Universal Robots PolyScope program: Presentacion.urp

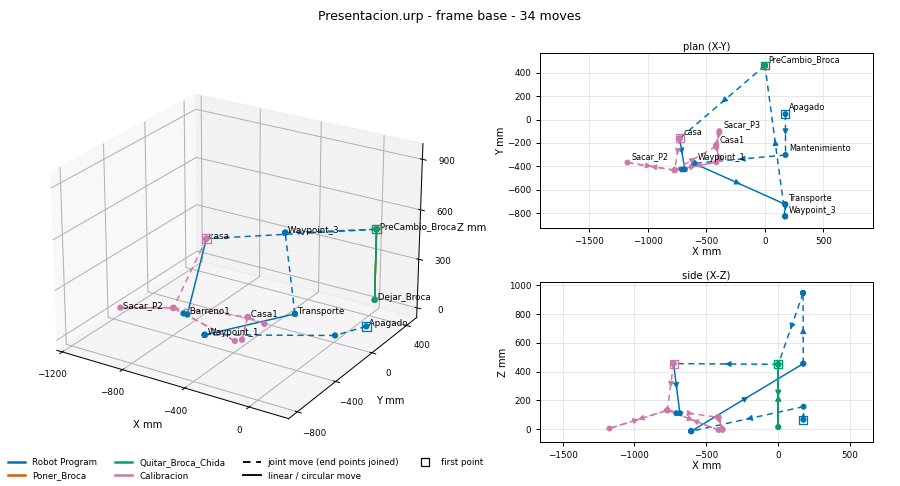
[picture p0: tool path of Presentacion.urp in frame base, 34 of 69 moves have a stored position in this frame; points joined in program order, loops and branches not executed]
Program Presentacion (installation=instalacion_derecha_10_MAR_21 directory=/programs/Presentacion createdIn=5.6.0.90886 lastSavedIn=5.6.0.90886 robotSerialNumber=20195001785)
Calibrated DH parameters: a=[0.000107, -0.568984, -0.552934, -0.00001, -0.000063, 0]; d=[0.180718, -257.998067, 200.685024, 57.48776, 0.119923, 0.115353]; alpha=[1.571119, 0.000876, -0.002498, 1.571178, -1.570523, 0]; deltaTheta=[0, -0.378191, 0.631587, -0.253396, 0, 0]
Robot Program (runOnlyOnce=false)
  MoveJ speed 60 deg/s, acceleration 80 deg/s^2 (useActiveTCP=true) feature=Base
    Waypoint Apagado: TCP in base x=175.753 y=46.675 z=64.304 mm, rx=-1.7747 ry=0.1396 rz=0.1139 rad; joints [90.002, -90.002, 153.585, 15, 89.999, 0.002] deg; TCP offset x=0.411 y=-218.298 z=37.994 mm, rx=1.558 ry=-0.1255 rz=0.1212 rad
    Waypoint Mantenimiento: TCP in base x=176.923 y=-302.82 z=155.559 mm, rx=0.3579 ry=-0.0299 rz=0.1455 rad; joints [90.14, -9.678, 128.928, 81.812, 89.499, -0.139] deg; TCP offset x=0.411 y=-218.298 z=37.994 mm, rx=1.558 ry=-0.1255 rz=0.1212 rad
  Folder Variables
    muestras := 3
    muestrasTomadas := 0
    alpha := 0
    P1 := p[0,0,0,0,0,0]
    P2 := p[0,0,0,0,0,0]
    P3 := p[0,0,0,0,0,0]
    P4 := p[0,0,0,0,0,0]
    Coordenada := p[0,0,0,0,0,0]
    MoveJ speed 60 deg/s, acceleration 80 deg/s^2 (useActiveTCP=true) feature=Base
      Loop Forever
        Waypoint Waypoint_1: TCP in base x=-604.792 y=-374.483 z=-15.265 mm, rx=2.0075 ry=-2.3999 rz=-0.0198 rad; joints [22.691, -71.513, 121.887, -50.957, 113.675, -0.127] deg; TCP offset x=0.411 y=-218.298 z=37.994 mm, rx=1.558 ry=-0.1255 rz=0.1212 rad
        Waypoint Waypoint_2: TCP in base x=-604.92 y=-374.48 z=-15.28 mm, rx=2.0074 ry=-2.4 rz=-0.0198 rad; joints [22.686, -71.504, 121.876, -50.954, 113.672, -0.127] deg
        var_7 := pose_dist(Waypoint_1, Waypoint_2)
      Waypoint Waypoint_1 referenceName=Waypoint_1: TCP in base x=-604.792 y=-374.483 z=-15.265 mm, rx=2.0075 ry=-2.3999 rz=-0.0198 rad; joints [22.691, -71.513, 121.887, -50.957, 113.675, -0.127] deg
      Waypoint Waypoint_2 referenceName=Waypoint_2: TCP in base x=-604.92 y=-374.48 z=-15.28 mm, rx=2.0074 ry=-2.4 rz=-0.0198 rad; joints [22.686, -71.504, 121.876, -50.954, 113.672, -0.127] deg
    pch_atual := get_actual_tcp_pose()
    Popup Message (haltProgram=false message=hi inputType=Variable) variable=pch_atual
  Folder Movimiento eje 7
    MoveL speed 250 mm/s, acceleration 1200 mm/s^2 (useActiveTCP=true) feature=Base
      Waypoint Transporte: TCP in base x=174.984 y=-724.59 z=455.169 mm, rx=3.1229 ry=-0.2484 rz=-0.0011 rad; joints [90, -90.004, 90.001, 0, 90, 0] deg; TCP offset x=0.411 y=-218.298 z=37.994 mm, rx=1.558 ry=-0.1255 rz=0.1212 rad
      Set DigitalOutput pin=postrnas_m187; digitalValue=1
      SuppressedNode
        Set ExpressionOutput pin=pos_2_mw3; expression=2
      num_barreno := str_cat("Barreno: ",1)
      var_6 := get_actual_tcp_pose()
      X_actual := str_cat("     X: ",var_6[0])
      Y_actual := str_cat("     Y: ",var_6[1])
      pos_barreno := str_cat(X_actual,Y_actual)
      Script: textmsg("------------------DAS LOG------------------")
      Script: textmsg(num_barreno,pos_barreno)
      Popup Warning (haltProgram=false message=hsjd inputType=Text)
  Folder Saludos
    MoveL speed 250 mm/s, acceleration 1200 mm/s^2 (useActiveTCP=true) feature=Base
      Waypoint Transporte: TCP in base x=174.984 y=-724.59 z=455.169 mm, rx=3.1229 ry=-0.2484 rz=-0.0011 rad; joints [90, -90.004, 90.001, 0, 90, 0] deg
      Set DigitalOutput pin=postrnas_m187; digitalValue=1
      SuppressedNode
        MoveJ speed 60 deg/s, acceleration 80 deg/s^2 (useActiveTCP=true) feature=Base
          Waypoint Casa: TCP in base x=728.924 y=-154.439 z=454.335 mm, rx=2.3654 ry=2.0675 rz=0 rad; joints [1.567, -90.267, -89.594, -180.639, -89.764, 0.039] deg
      MoveJ speed 60 deg/s, acceleration 80 deg/s^2 (useActiveTCP=true) feature=Base
        SuppressedNode
          Waypoint Waypoint_1: TCP in base x=65.093 y=-826.886 z=901.889 mm, rx=1.4338 ry=-0.7424 rz=0.7302 rad; joints [89.992, -97.74, 97.176, -89.444, 134.994, 0.001] deg
        Set DigitalOutput pin=postrnas_m187; digitalValue=0
        Waypoint Waypoint_3: TCP in base x=173.453 y=-827.062 z=946.896 mm, rx=1.4805 ry=-0.6168 rz=0.6108 rad; joints [98.118, -94.832, 92.691, -93.201, 125.502, -9.597] deg
        SuppressedNode
          Waypoint Waypoint_5: TCP in base x=173.423 y=-741.68 z=946.84 mm, rx=1.2989 ry=-0.7251 rz=0.6034 rad; joints [102.47, -97.376, 99.801, -114.266, 126.347, -24.689] deg
      Loop Counting (count=15) loopVariable(name=Loop_1)
        MoveL speed 1500 mm/s, acceleration 2200 mm/s^2 (useActiveTCP=true) feature=Base
          SuppressedNode
            Waypoint Waypoint_1: motionParameters(blendRadius=0.05); TCP in base x=65.093 y=-826.886 z=901.889 mm, rx=1.4338 ry=-0.7424 rz=0.7302 rad; joints [89.992, -97.74, 97.176, -89.444, 134.994, 0.001] deg
          SuppressedNode
            Waypoint Waypoint_2: motionParameters(blendRadius=0.05); TCP in base x=281.914 y=-909.743 z=901.9 mm, rx=1.5058 ry=0.4887 rz=-0.49 rad; joints [89.998, -90.003, 89.996, -90, 45, 0.004] deg
          Waypoint Waypoint_3: TCP in base x=173.453 y=-827.062 z=946.896 mm, rx=1.4805 ry=-0.6168 rz=0.6108 rad; joints [98.118, -94.832, 92.691, -93.201, 125.502, -9.597] deg
          Waypoint Waypoint_4: TCP in base x=173.444 y=-827.101 z=946.817 mm, rx=1.4837 ry=0.6112 rz=-0.6169 rad; joints [78.227, -99.572, 95.233, -100.465, 37.264, 18.965] deg
          SuppressedNode
            Waypoint Waypoint_5: motionParameters(jointSpeed=1.047198 jointAcceleration=1.396263 cartesianSpeed=0.25 cartesianAcceleration=1.2); TCP in base x=173.423 y=-741.68 z=946.84 mm, rx=1.2989 ry=-0.7251 rz=0.6034 rad; joints [102.47, -97.376, 99.801, -114.266, 126.347, -24.689] deg
          SuppressedNode
            Waypoint Waypoint_6: motionParameters(jointSpeed=1.047198 jointAcceleration=1.396263 cartesianSpeed=0.25 cartesianAcceleration=1.2); TCP in base x=173.459 y=-827.104 z=946.825 mm, rx=1.6228 ry=0.6313 rz=-0.7589 rad; joints [80.134, -100.807, 88.516, -73.712, 30.209, 3.288] deg
        SuppressedNode
          Waypoint Waypoint_1: TCP in base x=-291.405 y=-499.146 z=911.663 mm, rx=1.27 ry=-0.6711 rz=0.7685 rad; joints [-90.912, -52.098, -119.496, -88.535, -44.817, 0.182] deg
        SuppressedNode
          Waypoint Waypoint_2: TCP in base x=-77.693 y=-536.254 z=818.128 mm, rx=1.4537 ry=0.4411 rz=-0.4893 rad; joints [-90.912, -53.514, -125.158, -87.62, -133.489, 0.185] deg
      Popup Message (haltProgram=false message=arranquesito inputType=Text)
  SuppressedNode
    Popup Message (haltProgram=false message=opsjd inputType=Text)
  SuppressedNode
    Folder Paro_Emergencia
      MoveJ speed 60 deg/s, acceleration 80 deg/s^2 (useActiveTCP=true) feature=Base
        Waypoint Waypoint_3: TCP in base x=-687.031 y=180.786 z=3.5 mm, rx=1.8753 ry=-2.5169 rz=0.0061 rad; joints [-178.733, -104.887, -123.784, -131.854, -81.244, 0.422] deg
      MoveL speed 250 mm/s, acceleration 1200 mm/s^2 (useActiveTCP=true) feature=Base
        Loop Forever
          Waypoint Waypoint_3: TCP in base x=-687.031 y=180.786 z=3.5 mm, rx=1.8753 ry=-2.5169 rz=0.0061 rad; joints [-178.733, -104.887, -123.784, -131.854, -81.244, 0.422] deg
          Waypoint Waypoint_4: TCP in base x=-687.031 y=-113.957 z=3.5 mm, rx=1.8753 ry=-2.5169 rz=0.0061 rad; joints [-147.777, -104.253, -124.677, -131.662, -50.29, 0.749] deg
  Folder Cambio_Brocas
    Loop Counting (count=1) loopVariable=Loop_1
      MoveJ speed 60 deg/s, acceleration 80 deg/s^2 (useActiveTCP=true) feature=Base
        SuppressedNode
          Waypoint Transporte: TCP in base x=174.984 y=-724.59 z=455.169 mm, rx=3.1229 ry=-0.2484 rz=-0.0011 rad; joints [90, -90.004, 90.001, 0, 90, 0] deg
        SuppressedNode
          Waypoint Casa: TCP in base x=728.924 y=-154.439 z=454.335 mm, rx=2.3654 ry=2.0675 rz=0 rad; joints [1.567, -90.267, -89.594, -180.639, -89.764, 0.039] deg
        SuppressedNode
          Waypoint Pre_Casa: TCP in base x=724.591 y=175.02 z=455.143 mm, rx=2.3854 ry=2.034 rz=0.009 rad; joints [180.002, -90.001, 89.999, 0.004, 90, 0.002] deg; TCP offset x=0.411 y=-218.298 z=37.994 mm, rx=1.558 ry=-0.1255 rz=0.1212 rad
        SuppressedNode
          Waypoint Waypoint_7: TCP in base x=327.444 y=571.558 z=453.852 mm, rx=2.3843 ry=2.0357 rz=0.0036 rad; joints [90, -90, -90, -180, 0, 0] deg; TCP offset x=0.411 y=-218.298 z=37.994 mm, rx=1.558 ry=-0.1255 rz=0.1212 rad
        Waypoint PreCambio_Broca: TCP in base x=0.946 y=461.694 z=450 mm, rx=-0.2787 ry=-3.1292 rz=0 rad; joints [124.465, -59.781, -112.137, -188.57, -54.361, 0.335] deg
        SuppressedNode
          Loop Counting (count=50) loopVariable(name=Loop_1)
            Call Poner_Broca
            Call Quitar_Broca_Chida
        Call Poner_Broca
  Folder Barrenado
    alpha := 0
    Loop Forever
      MoveJ speed 60 deg/s, acceleration 80 deg/s^2 (useActiveTCP=true) feature=Base
        Waypoint casa: TCP in base x=-727.761 y=-161.288 z=455.169 mm, rx=2.012 ry=-2.4053 rz=-0.0107 rad; joints [-1.081, -90.004, 90.001, 0, 90, 0] deg; TCP offset x=0.411 y=-218.298 z=37.994 mm, rx=1.558 ry=-0.1255 rz=0.1212 rad
        Call Calibracion
        Call GoNoGo
        MoveL speed 250 mm/s, acceleration 1200 mm/s^2 (useActiveTCP=true) feature=Base
          Waypoint Barreno1: TCP in base x=-683.897 y=-425.831 z=110.04 mm, rx=3.0978 ry=-0.4471 rz=-0.0122 rad; joints [216.485, -110.43, -101.989, -147.498, -136.182, -0.299] deg
          Waypoint Barreno2: TCP in base x=-709.31 y=-425.852 z=110.052 mm, rx=3.0978 ry=-0.4471 rz=-0.0123 rad; joints [215.28, -112.388, -99.127, -148.4, -137.383, -0.296] deg
          Loop Counting (count=2) loopVariable(name=Loop_9)
            If alpha≤16
              internos := interpolate_pose(Barreno1, Barreno2, alpha)
              bajada := p[0,0,-0.024,0,0,0]
              subida := p[0,0,0.024,0,0,0]
              Waypoint Waypoint (Variable): variable=internos
              MoveDirectionNode (selectedDirection=ZMinus)
                Until DISTANCE (allowActions=false deceleration=3 distanceNodeType=STOP) Distance=0.067; motionParameters(blendRadius=0)
              MoveDirectionNode (selectedDirection=ZMinus toolParams=0.0013, 2.0E-4)
                Until TOOL_CONTACT_DETECTION (allowActions=false retraction=0 decelerationAcceleration=9 decelerationAngularAcceleration=34.906585)
              Wait Sleep waitTime=0.3
              Set DigitalOutput pin=config_out[1]; digitalValue=1
              Wait Sleep waitTime=0.5
              Set DigitalOutput pin=config_out[1]; digitalValue=0
              MoveDirectionNode (selectedDirection=ZPlus)
                Until DISTANCE (allowActions=false deceleration=3 distanceNodeType=STOP) Distance=0.002; motionParameters(blendRadius=0)
              Wait Sleep waitTime=0.5
              Set DigitalOutput pin=config_out[1]; digitalValue=1
              Wait Sleep waitTime=0.3
              Loop Counting (count=1) loopVariable(name=Loop_6)
                bajar := pose_add(get_actual_tcp_pose(), bajada)
                Waypoint Waypoint (Variable): motionParameters(jointSpeed=1.047198 jointAcceleration=1.396263 cartesianSpeed=0.005 cartesianAcceleration=0.01); variable=bajar
                subir := pose_add(get_actual_tcp_pose(), subida)
                Waypoint Waypoint (Variable): motionParameters(jointSpeed=1.047198 jointAcceleration=1.396263 cartesianSpeed=0.02 cartesianAcceleration=0.02); variable=subir
                bajada := pose_add(bajada, p[0,0,-0.008,0,0,0])
                subida := pose_add(subida, p[0,0,0.008,0,0,0])
              Set DigitalOutput pin=config_out[1]; digitalValue=0
              MoveDirectionNode (selectedDirection=ZPlus)
                Until DISTANCE (allowActions=false deceleration=3 distanceNodeType=STOP) Distance=0.1; motionParameters(blendRadius=0)
              alpha := alpha+1
            Else 
              Popup Message (haltProgram=false message=linea barrenada inputType=Text)
              Call Quitar_Broca_Chida
              Popup Message (haltProgram=false message=fin inputType=Text)
        Call Quitar_Broca_Chida
        Call Poner_Broca
SubProgram -> Poner_Broca
SubProgram -> Quitar_Broca_Chida
SubProgram -> Calibracion
SubProgram -> GoNoGo
SubProgram Poner_Broca (keepSynchronizedWithDisk=false)
  Folder Poner_Broca
    Set DigitalOutput pin=ini_cambro_m289; digitalValue=0
    MoveL speed 250 mm/s, acceleration 1200 mm/s^2 (useActiveTCP=true) feature=Base
      Waypoint PreCambio_Broca: TCP in base x=0.946 y=461.694 z=450 mm, rx=-0.2787 ry=-3.1292 rz=0 rad; joints [124.465, -59.781, -112.137, -188.57, -54.361, 0.335] deg; TCP offset x=0.411 y=-218.298 z=37.994 mm, rx=1.558 ry=-0.1255 rz=0.1212 rad
      Waypoint Dejar_Broca: TCP in base x=0.946 y=461.694 z=13.784 mm, rx=-0.2787 ry=-3.1292 rz=0 rad; joints [124.423, -78.567, -149.823, -132.118, -54.538, 0.369] deg; TCP offset x=0.411 y=-218.298 z=37.994 mm, rx=1.558 ry=-0.1255 rz=0.1212 rad
    Set DigitalOutput pin=ini_cambro_m289; digitalValue=1
    Wait Sleep waitTime=3.8
    Set DigitalOutput pin=ini_cambro_m289; digitalValue=0
    Wait Sleep waitTime=0.5
    Wait DigitalInput pin=fciclocarr_m292; digitalValue=0
    Wait Sleep waitTime=0.5
    MoveL speed 250 mm/s, acceleration 1200 mm/s^2 (useActiveTCP=true) feature=Base
      Waypoint PreCambio_Broca: TCP in base x=0.946 y=461.694 z=450 mm, rx=-0.2787 ry=-3.1292 rz=0 rad; joints [124.465, -59.781, -112.137, -188.57, -54.361, 0.335] deg; TCP offset x=0.411 y=-218.298 z=37.994 mm, rx=1.558 ry=-0.1255 rz=0.1212 rad
      SuppressedNode
        MoveJ speed 60 deg/s, acceleration 80 deg/s^2 (useActiveTCP=true) feature=Base
          Waypoint casa: TCP in base x=-327.476 y=-571.536 z=453.871 mm, rx=2.0383 ry=-2.3875 rz=-0.0101 rad; joints [269.996, -89.998, -90, -179.999, 0, 0] deg; TCP offset x=0.411 y=-218.298 z=37.994 mm, rx=1.558 ry=-0.1255 rz=0.1212 rad
    SuppressedNode
      Popup Message (haltProgram=false message=kon inputType=Text)
SubProgram Quitar_Broca_Chida (keepSynchronizedWithDisk=false)
  Folder Quitar_Broca
    MoveJ speed 60 deg/s, acceleration 80 deg/s^2 (useActiveTCP=true) feature=Base
      SuppressedNode
        Waypoint casa: TCP in base x=-734.526 y=-232.925 z=166.215 mm, rx=3.0978 ry=-0.4471 rz=-0.0122 rad; joints [200.498, -107.87, -99.095, -152.973, -152.157, -0.273] deg
      Loop Counting (count=1) loopVariable(name=Loop_3)
        MoveL speed 250 mm/s, acceleration 1200 mm/s^2 (useActiveTCP=true) feature=Base
          SuppressedNode
            MoveJ speed 60 deg/s, acceleration 80 deg/s^2 (useActiveTCP=true) feature=Base
              Waypoint casa: TCP in base x=-327.476 y=-571.536 z=453.871 mm, rx=2.0383 ry=-2.3875 rz=-0.0101 rad; joints [269.996, -89.998, -90, -179.999, 0, 0] deg
          MoveDirectionNode (selectedDirection=ZPlus)
            Until DISTANCE (allowActions=false deceleration=3 distanceNodeType=STOP) Distance=0.1; motionParameters(blendRadius=0)
          MoveJ speed 60 deg/s, acceleration 80 deg/s^2 (useActiveTCP=true) feature=Base
            Waypoint PreCambio_Broca: TCP in base x=0.946 y=461.694 z=450 mm, rx=-0.2787 ry=-3.1292 rz=0 rad; joints [124.465, -59.781, -112.137, -188.57, -54.361, 0.335] deg; TCP offset x=0.411 y=-218.298 z=37.994 mm, rx=1.558 ry=-0.1255 rz=0.1212 rad
          Waypoint Dejar_Broca: motionParameters(jointSpeed=1.047198 jointAcceleration=1.396263 cartesianSpeed=0.15 cartesianAcceleration=0.2); TCP in base x=0.946 y=461.694 z=13.784 mm, rx=-0.2787 ry=-3.1292 rz=0 rad; joints [124.423, -78.567, -149.823, -132.118, -54.538, 0.369] deg; TCP offset x=0.411 y=-218.298 z=37.994 mm, rx=1.558 ry=-0.1255 rz=0.1212 rad
          Set DigitalOutput pin=outputbroc_m291; digitalValue=1
          Wait Sleep waitTime=0.5
          Set DigitalOutput pin=outputbroc_m291; digitalValue=0
          Wait Sleep waitTime=0.5
          Wait DigitalInput pin=fciclocarr_m292; digitalValue=0
          Wait Sleep waitTime=0.5
          SuppressedNode
            MoveDirectionNode (selectedDirection=ZPlus)
              Until DISTANCE (allowActions=false deceleration=3 distanceNodeType=STOP) Distance=0.5; motionParameters(blendRadius=0)
          Waypoint PreCambio_Broca: TCP in base x=0.946 y=461.694 z=450 mm, rx=-0.2787 ry=-3.1292 rz=0 rad; joints [124.465, -59.781, -112.137, -188.57, -54.361, 0.335] deg; TCP offset x=0.411 y=-218.298 z=37.994 mm, rx=1.558 ry=-0.1255 rz=0.1212 rad
          Set DigitalOutput pin=avancarrusel_m7; digitalValue=1
          Wait Sleep waitTime=1.1
          Set DigitalOutput pin=avancarrusel_m7; digitalValue=0
          SuppressedNode
            Popup Message (haltProgram=false message=kon inputType=Text)
SubProgram Calibracion (keepSynchronizedWithDisk=false)
  Folder Calibracion
    Folder Subvariables
      muestras := 1
      muestrasTomadas := 0
      P1 := p[0,0,0,0,0,0]
      P2 := p[0,0,0,0,0,0]
      P3 := p[0,0,0,0,0,0]
      P4 := p[0,0,0,0,0,0]
      rotaciones := p[0,0,0,0,0,0]
      PosFinal := p[0,0,0,0,0,0]
      m1 := 0
      m2 := 0
      b1 := 0
      b2 := 0
      Xd := 0
      Yd := 0
      Xp := 0
      Yp := 0
      Xfin := 0
      Yfin := 0
    SuppressedNode
      Folder plano mod
        Loop Forever
          MoveL speed 250 mm/s, acceleration 1200 mm/s^2 (useActiveTCP=true) feature=Plane_5
            Popup Message (haltProgram=false inputType=Variable) variable(featureName=Plane_5)
            Waypoint Waypoint_5: TCP in base x=-413.934 y=-364.729 z=55.217 mm, rx=2.0101 ry=-2.4031 rz=-0.0102 rad; joints [31.806, -89.454, 133.906, -44.626, 122.803, 0.104] deg; TCP offset x=0.411 y=-218.298 z=37.994 mm, rx=1.558 ry=-0.1255 rz=0.1212 rad; feature pose in base x=-414.632 y=-364.771 z=-8.601 mm, rx=0.0051 ry=-3.1307 rz=0.001 rad
            Waypoint Waypoint_6: TCP in base x=-770.877 y=-364.729 z=55.217 mm, rx=2.0101 ry=-2.4031 rz=-0.0102 rad; joints [16.666, -66.533, 104.244, -37.849, 107.67, 0.156] deg
            SuppressedNode
              Script: 
            Script file /programs/Presentacion/nivelacion.script
              | MoveJ
              |       Waypoint_5
              | 
              | Plane5_const = pose_trans(Plane5_const, p[-0.5,-0.25,0.1,2.010,-2.403,-0.010])
            Popup Message (haltProgram=false inputType=Variable) variable(featureName=Plane_5)
            Waypoint Waypoint_5: TCP in base x=-413.934 y=-364.729 z=55.217 mm, rx=2.0101 ry=-2.4031 rz=-0.0102 rad; joints [31.806, -89.454, 133.906, -44.626, 122.803, 0.104] deg
            Waypoint Waypoint_6: TCP in base x=-770.877 y=-364.729 z=55.217 mm, rx=2.0101 ry=-2.4031 rz=-0.0102 rad; joints [16.666, -66.533, 104.244, -37.849, 107.67, 0.156] deg
    Folder Nivelacion
      SuppressedNode
        MoveL speed 250 mm/s, acceleration 1200 mm/s^2 (useActiveTCP=true) feature=Base
          MoveDirectionNode (selectedDirection=ZPlus)
            Until DISTANCE (allowActions=false deceleration=3 distanceNodeType=STOP) Distance=0.1; motionParameters(blendRadius=0)
          MoveJ speed 60 deg/s, acceleration 80 deg/s^2 (useActiveTCP=true) feature=Base
            Waypoint casa: TCP in base x=-727.761 y=-161.288 z=455.169 mm, rx=2.012 ry=-2.4053 rz=-0.0107 rad; joints [-1.081, -90.004, 90.001, 0, 90, 0] deg; TCP offset x=0.411 y=-218.298 z=37.994 mm, rx=1.558 ry=-0.1255 rz=0.1212 rad
          MoveL speed 250 mm/s, acceleration 1200 mm/s^2 (useActiveTCP=true) feature=Base
            MoveJ speed 60 deg/s, acceleration 80 deg/s^2 (useActiveTCP=true) feature=Base
              Waypoint Casa2: TCP in base x=-771.172 y=-432.935 z=130.553 mm, rx=2.0075 ry=-2.3998 rz=-0.0199 rad; joints [21.893, -67.533, 96.816, -29.884, 112.905, -0.164] deg
            Folder P1
              Loop While (checkContinuously=false) expression=muestrasTomadas<muestras
                MoveJ speed 60 deg/s, acceleration 80 deg/s^2 (useActiveTCP=true) feature=Base
                  Waypoint Sacar_P1: motionParameters(jointSpeed=1.047198 jointAcceleration=1.396263 cartesianSpeed=0.1 cartesianAcceleration=0.15); TCP in base x=-414.596 y=-364.737 z=-6.973 mm, rx=2.0075 ry=-2.3998 rz=-0.0199 rad; joints [31.933, -83.207, 136.677, -54.117, 122.913, -0.246] deg; TCP offset x=0.411 y=-218.298 z=37.994 mm, rx=1.558 ry=-0.1255 rz=0.1212 rad
                  SuppressedNode
                    Waypoint Sacar_P5: TCP in base x=-414.62 y=-364.74 z=-8.63 mm, rx=2.0074 ry=-2.3998 rz=-0.0199 rad; joints [31.932, -83.024, 136.735, -54.36, 122.914, -0.245] deg
                Wait Sleep waitTime=0.5
                MoveDirectionNode (selectedDirection=ZMinus toolParams=0.0013, 2.0E-4)
                  Until TOOL_CONTACT_DETECTION (allowActions=false retraction=0 decelerationAcceleration=9 decelerationAngularAcceleration=34.906585)
                Wait Sleep waitTime=2
                P5 := pose_add(get_actual_tcp_pose(), P5)
                muestrasTomadas := muestrasTomadas+1
              muestrasTomadas := 0
              var_1 := (P5[0])/muestras
              var_2 := (P5[1])/muestras
              var_8 := (P5[2])/muestras
              rotaciones := get_actual_tcp_pose()
              var_3 := rotaciones[3]
              var_4 := rotaciones[4]
              var_5 := rotaciones[5]
              P5 := p[var_1,var_2,var_8,var_3,var_4,var_5]
            MoveJ speed 60 deg/s, acceleration 80 deg/s^2 (useActiveTCP=true) feature=Base
              Waypoint Casa2: TCP in base x=-771.172 y=-432.935 z=130.553 mm, rx=2.0075 ry=-2.3998 rz=-0.0199 rad; joints [21.893, -67.533, 96.816, -29.884, 112.905, -0.164] deg; TCP offset x=0.411 y=-218.298 z=37.994 mm, rx=1.558 ry=-0.1255 rz=0.1212 rad
            Folder P2
              Loop While (checkContinuously=false) expression=muestrasTomadas<muestras
                MoveJ speed 60 deg/s, acceleration 80 deg/s^2 (useActiveTCP=true) feature=Base
                  Waypoint Sacar_P2: TCP in base x=-1173.98 y=-367.222 z=3.642 mm, rx=2.0075 ry=-2.3998 rz=-0.0199 rad; joints [10.692, -31.748, 48.291, -17.094, 101.74, -0.036] deg; TCP offset x=0.411 y=-218.298 z=37.994 mm, rx=1.558 ry=-0.1255 rz=0.1212 rad
                  SuppressedNode
                    Waypoint Sacar_P6: TCP in base x=-1173.985 y=-367.26 z=-0.32 mm, rx=2.0075 ry=-2.3998 rz=-0.0199 rad; joints [10.694, -31.605, 48.427, -17.374, 101.738, -0.036] deg
                Wait Sleep waitTime=0.5
                MoveDirectionNode (selectedDirection=YPlus toolParams=0.0013, 2.0E-4)
                  Until TOOL_CONTACT_DETECTION (allowActions=false retraction=0 decelerationAcceleration=9 decelerationAngularAcceleration=34.906585)
                Wait Sleep waitTime=2
                P2 := pose_add(get_actual_tcp_pose(), P2)
                muestrasTomadas := muestrasTomadas+1
              muestrasTomadas := 0
              var_1 := (P2[0])/muestras
              var_2 := (P2[1])/muestras
              rotaciones := get_actual_tcp_pose()
              var_3 := rotaciones[3]
              var_4 := rotaciones[4]
              var_5 := rotaciones[5]
              P2 := p[var_1,var_2,-0.37,var_3,var_4,var_5]
            MoveJ speed 60 deg/s, acceleration 80 deg/s^2 (useActiveTCP=true) feature=Base
              Waypoint Casa2: TCP in base x=-771.172 y=-432.935 z=130.553 mm, rx=2.0075 ry=-2.3998 rz=-0.0199 rad; joints [21.893, -67.533, 96.816, -29.884, 112.905, -0.164] deg; TCP offset x=0.411 y=-218.298 z=37.994 mm, rx=1.558 ry=-0.1255 rz=0.1212 rad
            Folder m1
              var_1 := (P1[0])
              var_2 := (P1[1])
              var_3 := (P2[0])
              var_4 := (P2[1])
              m1 := (var_4-var_2)/(var_3-var_1)
            Folder b1
              b1 := ((m1*var_1)-var_2)*(-1)
            MoveJ speed 60 deg/s, acceleration 80 deg/s^2 (useActiveTCP=true) feature=Base
              Waypoint Casa1: TCP in base x=-397.714 y=-209.387 z=130.553 mm, rx=2.0075 ry=-2.3998 rz=-0.0199 rad; joints [8.28, -111.842, 141.427, -30.137, 99.306, -0.058] deg; TCP offset x=0.411 y=-218.298 z=37.994 mm, rx=1.558 ry=-0.1255 rz=0.1212 rad
            Folder P3
              Loop While (checkContinuously=false) expression=muestrasTomadas<muestras
                MoveJ speed 60 deg/s, acceleration 80 deg/s^2 (useActiveTCP=true) feature=Base
                  Waypoint Sacar_P3: motionParameters(jointSpeed=1.047198 jointAcceleration=1.396263 cartesianSpeed=0.1 cartesianAcceleration=0.15); TCP in base x=-389.257 y=-99.052 z=-5.952 mm, rx=2.0075 ry=-2.3998 rz=-0.0199 rad; joints [-19.785, -107.959, 157.177, -49.758, 71.211, 0.249] deg
                  SuppressedNode
                    Waypoint Sacar_P7: TCP in base x=-389.26 y=-99.06 z=-9.06 mm, rx=2.0075 ry=-2.3998 rz=-0.02 rad; joints [-19.783, -107.388, 157.374, -50.532, 71.212, 0.252] deg
                Wait Sleep waitTime=0.5
                MoveDirectionNode (selectedDirection=XPlus toolParams=0.0013, 2.0E-4)
                  Until TOOL_CONTACT_DETECTION (allowActions=false retraction=0 decelerationAcceleration=9 decelerationAngularAcceleration=34.906585)
                Wait Sleep waitTime=2
                P3 := pose_add(get_actual_tcp_pose(), P3)
                muestrasTomadas := muestrasTomadas+1
              muestrasTomadas := 0
              var_1 := (P3[0])/muestras
              var_2 := (P3[1])/muestras
              rotaciones := get_actual_tcp_pose()
              var_3 := rotaciones[3]
              var_4 := rotaciones[4]
              var_5 := rotaciones[5]
              P3 := p[var_1,var_2,-0.37,var_3,var_4,var_5]
            MoveJ speed 60 deg/s, acceleration 80 deg/s^2 (useActiveTCP=true) feature=Base
              Waypoint Casa1: TCP in base x=-397.714 y=-209.387 z=130.553 mm, rx=2.0075 ry=-2.3998 rz=-0.0199 rad; joints [8.28, -111.842, 141.427, -30.137, 99.306, -0.058] deg
            Folder P4
              Loop While (checkContinuously=false) expression=muestrasTomadas<muestras
                MoveJ speed 60 deg/s, acceleration 80 deg/s^2 (useActiveTCP=true) feature=Base
                  Waypoint Sacar_P4: motionParameters(jointSpeed=1.047198 jointAcceleration=1.396263 cartesianSpeed=0.1 cartesianAcceleration=0.15); TCP in base x=-387.922 y=-336.637 z=-4.002 mm, rx=2.0075 ry=-2.3998 rz=-0.0199 rad; joints [30.437, -87.075, 140.636, -54.198, 121.418, -0.23] deg
                Wait Sleep waitTime=0.5
                MoveDirectionNode (selectedDirection=XPlus toolParams=0.0013, 2.0E-4)
                  Until TOOL_CONTACT_DETECTION (allowActions=false retraction=0 decelerationAcceleration=9 decelerationAngularAcceleration=34.906585)
                Wait Sleep waitTime=2
                P4 := pose_add(get_actual_tcp_pose(), P4)
                muestrasTomadas := muestrasTomadas+1
              muestrasTomadas := 0
              var_1 := (P4[0])/muestras
              var_2 := (P4[1])/muestras
              rotaciones := get_actual_tcp_pose()
              var_3 := rotaciones[3]
              var_4 := rotaciones[4]
              var_5 := rotaciones[5]
              P4 := p[var_1,var_2,-0.37,var_3,var_4,var_5]
            MoveJ speed 60 deg/s, acceleration 80 deg/s^2 (useActiveTCP=true) feature=Base
              Waypoint Casa1: TCP in base x=-397.714 y=-209.387 z=130.553 mm, rx=2.0075 ry=-2.3998 rz=-0.0199 rad; joints [8.28, -111.842, 141.427, -30.137, 99.306, -0.058] deg
            Folder m2
              var_1 := (P3[0])
              var_2 := (P3[1])
              var_3 := (P4[0])
              var_4 := (P4[1])
              m2 := (var_4-var_2)/(var_3-var_1)
            Folder b2
              b2 := ((m2*var_1)-var_2)*(-1)
            Folder Xd y Yd
              Xd := (b2-b1)/(m1-m2)
              Yd := (m1*Xd)+b1
            Folder Xp y Yp
              Xp := (1)/(sqrt((m1*m1)+1))
              Yp := (m2)/(sqrt((m2*m2)+1))
            Folder Origen
              Xfin := ((0*Xp)-(Xd)-(0*(1/m2)))*(-1)
              Yfin := ((0*Yp)-(Yd)+(0*m1))*(-1)
              rotaciones := get_actual_tcp_pose()
              var_3 := rotaciones[3]
              var_4 := rotaciones[4]
              var_5 := rotaciones[5]
              PosFinal := p[Xfin+0.00208915,Yfin+0.00208915,0.11,var_3,var_4,var_5]
            MoveJ speed 60 deg/s, acceleration 80 deg/s^2 (useActiveTCP=true) feature=Base
              Waypoint Waypoint (Variable): motionParameters(jointSpeed=1.047198 jointAcceleration=1.396263 cartesianSpeed=0.15 cartesianAcceleration=0.2); variable=PosFinal
            MoveDirectionNode (selectedDirection=ZPlus)
              Until DISTANCE (allowActions=false deceleration=3 distanceNodeType=STOP) Distance=0.1; motionParameters(blendRadius=0)
            MoveJ speed 60 deg/s, acceleration 80 deg/s^2 (useActiveTCP=true) feature=Base
              Waypoint Casa2: TCP in base x=-771.172 y=-432.935 z=130.553 mm, rx=2.0075 ry=-2.3998 rz=-0.0199 rad; joints [21.893, -67.533, 96.816, -29.884, 112.905, -0.164] deg; TCP offset x=0.411 y=-218.298 z=37.994 mm, rx=1.558 ry=-0.1255 rz=0.1212 rad
            Folder Linea1
              Folder Buje1
                Xfin := ((0.09525*Xp)-(Xd)-(-0.0127*(1/m2)))*(-1)
                Yfin := ((-0.0127*Yp)-(Yd)+(0.09525*m1))*(-1)
                rotaciones := get_actual_tcp_pose()
                var_3 := rotaciones[3]
                var_4 := rotaciones[4]
                var_5 := rotaciones[5]
                PosFinal := p[Xfin+0.00208915,Yfin+0.00208915,0.03,var_3,var_4,var_5]
                MoveL speed 250 mm/s, acceleration 1200 mm/s^2 (useActiveTCP=true) feature=Base
                  MoveJ speed 60 deg/s, acceleration 80 deg/s^2 (useActiveTCP=true) feature=Base
                    Waypoint Waypoint (Variable): motionParameters(jointSpeed=1.047198 jointAcceleration=1.396263 cartesianSpeed=0.15 cartesianAcceleration=0.2); variable=PosFinal
                  MoveDirectionNode (selectedDirection=ZMinus toolParams=0.02, 0.02)
                    Until DISTANCE (allowActions=false deceleration=3 distanceNodeType=STOP) Distance=0.035; motionParameters(blendRadius=0)
                  MoveDirectionNode (selectedDirection=ZPlus toolParams=0.02, 0.02)
                    Until DISTANCE (allowActions=false deceleration=3 distanceNodeType=STOP) Distance=0.035; motionParameters(blendRadius=0)
              Folder Buje2
                Xfin := ((0.12065*Xp)-(Xd)-(-0.0127*(1/m2)))*(-1)
                Yfin := ((-0.0127*Yp)-(Yd)+(0.12065*m1))*(-1)
                rotaciones := get_actual_tcp_pose()
                var_3 := rotaciones[3]
                var_4 := rotaciones[4]
                var_5 := rotaciones[5]
                PosFinal := p[Xfin+0.00208915,Yfin+0.00208915,0.03,var_3,var_4,var_5]
                MoveL speed 250 mm/s, acceleration 1200 mm/s^2 (useActiveTCP=true) feature=Base
                  MoveJ speed 60 deg/s, acceleration 80 deg/s^2 (useActiveTCP=true) feature=Base
                    Waypoint Waypoint (Variable): motionParameters(jointSpeed=1.047198 jointAcceleration=1.396263 cartesianSpeed=0.15 cartesianAcceleration=0.2); variable=PosFinal
                  MoveDirectionNode (selectedDirection=ZMinus toolParams=0.02, 0.02)
                    Until DISTANCE (allowActions=false deceleration=3 distanceNodeType=STOP) Distance=0.035; motionParameters(blendRadius=0)
                  MoveDirectionNode (selectedDirection=ZPlus toolParams=0.02, 0.02)
                    Until DISTANCE (allowActions=false deceleration=3 distanceNodeType=STOP) Distance=0.035; motionParameters(blendRadius=0)
              Folder Buje3
                Xfin := ((0.14605*Xp)-(Xd)-(-0.0127*(1/m2)))*(-1)
                Yfin := ((-0.0127*Yp)-(Yd)+(0.14605*m1))*(-1)
                rotaciones := get_actual_tcp_pose()
                var_3 := rotaciones[3]
                var_4 := rotaciones[4]
                var_5 := rotaciones[5]
                PosFinal := p[Xfin+0.00208915,Yfin+0.00208915,0.03,var_3,var_4,var_5]
                MoveL speed 250 mm/s, acceleration 1200 mm/s^2 (useActiveTCP=true) feature=Base
                  MoveJ speed 60 deg/s, acceleration 80 deg/s^2 (useActiveTCP=true) feature=Base
                    Waypoint Waypoint (Variable): motionParameters(jointSpeed=1.047198 jointAcceleration=1.396263 cartesianSpeed=0.15 cartesianAcceleration=0.2); variable=PosFinal
                  MoveDirectionNode (selectedDirection=ZMinus toolParams=0.02, 0.02)
                    Until DISTANCE (allowActions=false deceleration=3 distanceNodeType=STOP) Distance=0.035; motionParameters(blendRadius=0)
                  MoveDirectionNode (selectedDirection=ZPlus toolParams=0.02, 0.02)
                    Until DISTANCE (allowActions=false deceleration=3 distanceNodeType=STOP) Distance=0.035; motionParameters(blendRadius=0)
              SuppressedNode
                Folder Buje4
                  Xfin := ((0.17145*Xp)-(Xd)-(-0.0127*(1/m2)))*(-1)
                  Yfin := ((-0.0127*Yp)-(Yd)+(0.17145*m1))*(-1)
                  rotaciones := get_actual_tcp_pose()
                  var_3 := rotaciones[3]
                  var_4 := rotaciones[4]
                  var_5 := rotaciones[5]
                  PosFinal := p[Xfin+0.00208915,Yfin+0.00208915,0.03,var_3,var_4,var_5]
                  MoveL speed 250 mm/s, acceleration 1200 mm/s^2 (useActiveTCP=true) feature=Base
                    MoveJ speed 60 deg/s, acceleration 80 deg/s^2 (useActiveTCP=true) feature=Base
                      Waypoint Waypoint (Variable): motionParameters(jointSpeed=1.047198 jointAcceleration=1.396263 cartesianSpeed=0.15 cartesianAcceleration=0.2); variable=PosFinal
                    MoveDirectionNode (selectedDirection=ZMinus toolParams=0.02, 0.02)
                      Until DISTANCE (allowActions=false deceleration=3 distanceNodeType=STOP) Distance=0.035; motionParameters(blendRadius=0)
                    MoveDirectionNode (selectedDirection=ZPlus toolParams=0.02, 0.02)
                      Until DISTANCE (allowActions=false deceleration=3 distanceNodeType=STOP) Distance=0.035; motionParameters(blendRadius=0)
              SuppressedNode
                Folder Buje5
                  Xfin := ((0.19685*Xp)-(Xd)-(-0.0127*(1/m2)))*(-1)
                  Yfin := ((-0.0127*Yp)-(Yd)+(0.19685*m1))*(-1)
                  rotaciones := get_actual_tcp_pose()
                  var_3 := rotaciones[3]
                  var_4 := rotaciones[4]
                  var_5 := rotaciones[5]
                  PosFinal := p[Xfin+0.00208915,Yfin+0.00208915,0.03,var_3,var_4,var_5]
                  MoveL speed 250 mm/s, acceleration 1200 mm/s^2 (useActiveTCP=true) feature=Base
                    MoveJ speed 60 deg/s, acceleration 80 deg/s^2 (useActiveTCP=true) feature=Base
                      Waypoint Waypoint (Variable): motionParameters(jointSpeed=1.047198 jointAcceleration=1.396263 cartesianSpeed=0.15 cartesianAcceleration=0.2); variable=PosFinal
                    MoveDirectionNode (selectedDirection=ZMinus toolParams=0.02, 0.02)
                      Until DISTANCE (allowActions=false deceleration=3 distanceNodeType=STOP) Distance=0.035; motionParameters(blendRadius=0)
                    MoveDirectionNode (selectedDirection=ZPlus toolParams=0.02, 0.02)
                      Until DISTANCE (allowActions=false deceleration=3 distanceNodeType=STOP) Distance=0.035; motionParameters(blendRadius=0)
              SuppressedNode
                Folder Buje6
                  Xfin := ((0.22225*Xp)-(Xd)-(-0.0127*(1/m2)))*(-1)
                  Yfin := ((-0.0127*Yp)-(Yd)+(0.22225*m1))*(-1)
                  rotaciones := get_actual_tcp_pose()
                  var_3 := rotaciones[3]
                  var_4 := rotaciones[4]
                  var_5 := rotaciones[5]
                  PosFinal := p[Xfin+0.00208915,Yfin+0.00208915,0.03,var_3,var_4,var_5]
                  MoveL speed 250 mm/s, acceleration 1200 mm/s^2 (useActiveTCP=true) feature=Base
                    MoveJ speed 60 deg/s, acceleration 80 deg/s^2 (useActiveTCP=true) feature=Base
                      Waypoint Waypoint (Variable): motionParameters(jointSpeed=1.047198 jointAcceleration=1.396263 cartesianSpeed=0.15 cartesianAcceleration=0.2); variable=PosFinal
                    MoveDirectionNode (selectedDirection=ZMinus toolParams=0.02, 0.02)
                      Until DISTANCE (allowActions=false deceleration=3 distanceNodeType=STOP) Distance=0.035; motionParameters(blendRadius=0)
                    MoveDirectionNode (selectedDirection=ZPlus toolParams=0.02, 0.02)
                      Until DISTANCE (allowActions=false deceleration=3 distanceNodeType=STOP) Distance=0.035; motionParameters(blendRadius=0)
              SuppressedNode
                Folder Buje7
                  Xfin := ((0.24765*Xp)-(Xd)-(-0.0127*(1/m2)))*(-1)
                  Yfin := ((-0.0127*Yp)-(Yd)+(0.24765*m1))*(-1)
                  rotaciones := get_actual_tcp_pose()
                  var_3 := rotaciones[3]
                  var_4 := rotaciones[4]
                  var_5 := rotaciones[5]
                  PosFinal := p[Xfin+0.00208915,Yfin+0.00208915,0.03,var_3,var_4,var_5]
                  MoveL speed 250 mm/s, acceleration 1200 mm/s^2 (useActiveTCP=true) feature=Base
                    MoveJ speed 60 deg/s, acceleration 80 deg/s^2 (useActiveTCP=true) feature=Base
                      Waypoint Waypoint (Variable): motionParameters(jointSpeed=1.047198 jointAcceleration=1.396263 cartesianSpeed=0.15 cartesianAcceleration=0.2); variable=PosFinal
                    MoveDirectionNode (selectedDirection=ZMinus toolParams=0.02, 0.02)
                      Until DISTANCE (allowActions=false deceleration=3 distanceNodeType=STOP) Distance=0.035; motionParameters(blendRadius=0)
                    MoveDirectionNode (selectedDirection=ZPlus toolParams=0.02, 0.02)
                      Until DISTANCE (allowActions=false deceleration=3 distanceNodeType=STOP) Distance=0.035; motionParameters(blendRadius=0)
              SuppressedNode
                Folder Buje8
                  Xfin := ((0.27305*Xp)-(Xd)-(-0.0127*(1/m2)))*(-1)
                  Yfin := ((-0.0127*Yp)-(Yd)+(0.27305*m1))*(-1)
                  rotaciones := get_actual_tcp_pose()
                  var_3 := rotaciones[3]
                  var_4 := rotaciones[4]
                  var_5 := rotaciones[5]
                  PosFinal := p[Xfin+0.00208915,Yfin+0.00208915,0.03,var_3,var_4,var_5]
                  MoveL speed 250 mm/s, acceleration 1200 mm/s^2 (useActiveTCP=true) feature=Base
                    MoveJ speed 60 deg/s, acceleration 80 deg/s^2 (useActiveTCP=true) feature=Base
                      Waypoint Waypoint (Variable): motionParameters(jointSpeed=1.047198 jointAcceleration=1.396263 cartesianSpeed=0.15 cartesianAcceleration=0.2); variable=PosFinal
                    MoveDirectionNode (selectedDirection=ZMinus toolParams=0.02, 0.02)
                      Until DISTANCE (allowActions=false deceleration=3 distanceNodeType=STOP) Distance=0.035; motionParameters(blendRadius=0)
                    MoveDirectionNode (selectedDirection=ZPlus toolParams=0.02, 0.02)
                      Until DISTANCE (allowActions=false deceleration=3 distanceNodeType=STOP) Distance=0.035; motionParameters(blendRadius=0)
              SuppressedNode
                Folder Buje9
                  Xfin := ((0.29845*Xp)-(Xd)-(-0.0127*(1/m2)))*(-1)
                  Yfin := ((-0.0127*Yp)-(Yd)+(0.29845*m1))*(-1)
                  rotaciones := get_actual_tcp_pose()
                  var_3 := rotaciones[3]
                  var_4 := rotaciones[4]
                  var_5 := rotaciones[5]
                  PosFinal := p[Xfin+0.00208915,Yfin+0.00208915,0.03,var_3,var_4,var_5]
                  MoveL speed 250 mm/s, acceleration 1200 mm/s^2 (useActiveTCP=true) feature=Base
                    MoveJ speed 60 deg/s, acceleration 80 deg/s^2 (useActiveTCP=true) feature=Base
                      Waypoint Waypoint (Variable): motionParameters(jointSpeed=1.047198 jointAcceleration=1.396263 cartesianSpeed=0.15 cartesianAcceleration=0.2); variable=PosFinal
                    MoveDirectionNode (selectedDirection=ZMinus toolParams=0.02, 0.02)
                      Until DISTANCE (allowActions=false deceleration=3 distanceNodeType=STOP) Distance=0.035; motionParameters(blendRadius=0)
                    MoveDirectionNode (selectedDirection=ZPlus toolParams=0.02, 0.02)
                      Until DISTANCE (allowActions=false deceleration=3 distanceNodeType=STOP) Distance=0.035; motionParameters(blendRadius=0)
              SuppressedNode
                Folder Buje10
                  Xfin := ((0.32385*Xp)-(Xd)-(-0.0127*(1/m2)))*(-1)
                  Yfin := ((-0.0127*Yp)-(Yd)+(0.32385*m1))*(-1)
                  rotaciones := get_actual_tcp_pose()
                  var_3 := rotaciones[3]
                  var_4 := rotaciones[4]
                  var_5 := rotaciones[5]
                  PosFinal := p[Xfin+0.00208915,Yfin+0.00208915,0.03,var_3,var_4,var_5]
                  MoveL speed 250 mm/s, acceleration 1200 mm/s^2 (useActiveTCP=true) feature=Base
                    MoveJ speed 60 deg/s, acceleration 80 deg/s^2 (useActiveTCP=true) feature=Base
                      Waypoint Waypoint (Variable): motionParameters(jointSpeed=1.047198 jointAcceleration=1.396263 cartesianSpeed=0.15 cartesianAcceleration=0.2); variable=PosFinal
                    MoveDirectionNode (selectedDirection=ZMinus toolParams=0.02, 0.02)
                      Until DISTANCE (allowActions=false deceleration=3 distanceNodeType=STOP) Distance=0.035; motionParameters(blendRadius=0)
                    MoveDirectionNode (selectedDirection=ZPlus toolParams=0.02, 0.02)
                      Until DISTANCE (allowActions=false deceleration=3 distanceNodeType=STOP) Distance=0.035; motionParameters(blendRadius=0)
              SuppressedNode
                Folder Buje11
                  Xfin := ((0.34925*Xp)-(Xd)-(-0.0127*(1/m2)))*(-1)
                  Yfin := ((-0.0127*Yp)-(Yd)+(0.34925*m1))*(-1)
                  rotaciones := get_actual_tcp_pose()
                  var_3 := rotaciones[3]
                  var_4 := rotaciones[4]
                  var_5 := rotaciones[5]
                  PosFinal := p[Xfin+0.00208915,Yfin+0.00208915,0.03,var_3,var_4,var_5]
                  MoveL speed 250 mm/s, acceleration 1200 mm/s^2 (useActiveTCP=true) feature=Base
                    MoveJ speed 60 deg/s, acceleration 80 deg/s^2 (useActiveTCP=true) feature=Base
                      Waypoint Waypoint (Variable): motionParameters(jointSpeed=1.047198 jointAcceleration=1.396263 cartesianSpeed=0.15 cartesianAcceleration=0.2); variable=PosFinal
                    MoveDirectionNode (selectedDirection=ZMinus toolParams=0.02, 0.02)
                      Until DISTANCE (allowActions=false deceleration=3 distanceNodeType=STOP) Distance=0.035; motionParameters(blendRadius=0)
                    MoveDirectionNode (selectedDirection=ZPlus toolParams=0.02, 0.02)
                      Until DISTANCE (allowActions=false deceleration=3 distanceNodeType=STOP) Distance=0.035; motionParameters(blendRadius=0)
              SuppressedNode
                Folder Buje12
                  Xfin := ((0.37465*Xp)-(Xd)-(-0.0127*(1/m2)))*(-1)
                  Yfin := ((-0.0127*Yp)-(Yd)+(0.37465*m1))*(-1)
                  rotaciones := get_actual_tcp_pose()
                  var_3 := rotaciones[3]
                  var_4 := rotaciones[4]
                  var_5 := rotaciones[5]
                  PosFinal := p[Xfin+0.00208915,Yfin+0.00208915,0.03,var_3,var_4,var_5]
                  MoveL speed 250 mm/s, acceleration 1200 mm/s^2 (useActiveTCP=true) feature=Base
                    MoveJ speed 60 deg/s, acceleration 80 deg/s^2 (useActiveTCP=true) feature=Base
                      Waypoint Waypoint (Variable): motionParameters(jointSpeed=1.047198 jointAcceleration=1.396263 cartesianSpeed=0.15 cartesianAcceleration=0.2); variable=PosFinal
                    MoveDirectionNode (selectedDirection=ZMinus toolParams=0.02, 0.02)
                      Until DISTANCE (allowActions=false deceleration=3 distanceNodeType=STOP) Distance=0.035; motionParameters(blendRadius=0)
                    MoveDirectionNode (selectedDirection=ZPlus toolParams=0.02, 0.02)
                      Until DISTANCE (allowActions=false deceleration=3 distanceNodeType=STOP) Distance=0.035; motionParameters(blendRadius=0)
              SuppressedNode
                Folder Buje13
                  Xfin := ((0.40005*Xp)-(Xd)-(-0.0127*(1/m2)))*(-1)
                  Yfin := ((-0.0127*Yp)-(Yd)+(0.40005*m1))*(-1)
                  rotaciones := get_actual_tcp_pose()
                  var_3 := rotaciones[3]
                  var_4 := rotaciones[4]
                  var_5 := rotaciones[5]
                  PosFinal := p[Xfin+0.00208915,Yfin+0.00208915,0.03,var_3,var_4,var_5]
                  MoveL speed 250 mm/s, acceleration 1200 mm/s^2 (useActiveTCP=true) feature=Base
                    MoveJ speed 60 deg/s, acceleration 80 deg/s^2 (useActiveTCP=true) feature=Base
                      Waypoint Waypoint (Variable): motionParameters(jointSpeed=1.047198 jointAcceleration=1.396263 cartesianSpeed=0.15 cartesianAcceleration=0.2); variable=PosFinal
                    MoveDirectionNode (selectedDirection=ZMinus toolParams=0.02, 0.02)
                      Until DISTANCE (allowActions=false deceleration=3 distanceNodeType=STOP) Distance=0.035; motionParameters(blendRadius=0)
                    MoveDirectionNode (selectedDirection=ZPlus toolParams=0.02, 0.02)
                      Until DISTANCE (allowActions=false deceleration=3 distanceNodeType=STOP) Distance=0.035; motionParameters(blendRadius=0)
              SuppressedNode
                Folder Buje14
                  Xfin := ((0.42545*Xp)-(Xd)-(-0.0127*(1/m2)))*(-1)
                  Yfin := ((-0.0127*Yp)-(Yd)+(0.42545*m1))*(-1)
                  rotaciones := get_actual_tcp_pose()
                  var_3 := rotaciones[3]
                  var_4 := rotaciones[4]
                  var_5 := rotaciones[5]
                  PosFinal := p[Xfin+0.00208915,Yfin+0.00208915,0.03,var_3,var_4,var_5]
                  MoveL speed 250 mm/s, acceleration 1200 mm/s^2 (useActiveTCP=true) feature=Base
                    MoveJ speed 60 deg/s, acceleration 80 deg/s^2 (useActiveTCP=true) feature=Base
                      Waypoint Waypoint (Variable): motionParameters(jointSpeed=1.047198 jointAcceleration=1.396263 cartesianSpeed=0.15 cartesianAcceleration=0.2); variable=PosFinal
                    MoveDirectionNode (selectedDirection=ZMinus toolParams=0.02, 0.02)
                      Until DISTANCE (allowActions=false deceleration=3 distanceNodeType=STOP) Distance=0.035; motionParameters(blendRadius=0)
                    MoveDirectionNode (selectedDirection=ZPlus toolParams=0.02, 0.02)
                      Until DISTANCE (allowActions=false deceleration=3 distanceNodeType=STOP) Distance=0.035; motionParameters(blendRadius=0)
              SuppressedNode
                Folder Buje15
                  Xfin := ((0.45085*Xp)-(Xd)-(-0.0127*(1/m2)))*(-1)
                  Yfin := ((-0.0127*Yp)-(Yd)+(0.45085*m1))*(-1)
                  rotaciones := get_actual_tcp_pose()
                  var_3 := rotaciones[3]
                  var_4 := rotaciones[4]
                  var_5 := rotaciones[5]
                  PosFinal := p[Xfin+0.00208915,Yfin+0.00208915,0.03,var_3,var_4,var_5]
                  MoveL speed 250 mm/s, acceleration 1200 mm/s^2 (useActiveTCP=true) feature=Base
                    MoveJ speed 60 deg/s, acceleration 80 deg/s^2 (useActiveTCP=true) feature=Base
                      Waypoint Waypoint (Variable): motionParameters(jointSpeed=1.047198 jointAcceleration=1.396263 cartesianSpeed=0.15 cartesianAcceleration=0.2); variable=PosFinal
                    MoveDirectionNode (selectedDirection=ZMinus toolParams=0.02, 0.02)
                      Until DISTANCE (allowActions=false deceleration=3 distanceNodeType=STOP) Distance=0.035; motionParameters(blendRadius=0)
                    MoveDirectionNode (selectedDirection=ZPlus toolParams=0.02, 0.02)
                      Until DISTANCE (allowActions=false deceleration=3 distanceNodeType=STOP) Distance=0.035; motionParameters(blendRadius=0)
              SuppressedNode
                Folder Buje16
                  Xfin := ((0.47625*Xp)-(Xd)-(-0.0127*(1/m2)))*(-1)
                  Yfin := ((-0.0127*Yp)-(Yd)+(0.47625*m1))*(-1)
                  rotaciones := get_actual_tcp_pose()
                  var_3 := rotaciones[3]
                  var_4 := rotaciones[4]
                  var_5 := rotaciones[5]
                  PosFinal := p[Xfin+0.00208915,Yfin+0.00208915,0.03,var_3,var_4,var_5]
                  MoveL speed 250 mm/s, acceleration 1200 mm/s^2 (useActiveTCP=true) feature=Base
                    MoveJ speed 60 deg/s, acceleration 80 deg/s^2 (useActiveTCP=true) feature=Base
                      Waypoint Waypoint (Variable): motionParameters(jointSpeed=1.047198 jointAcceleration=1.396263 cartesianSpeed=0.15 cartesianAcceleration=0.2); variable=PosFinal
                    MoveDirectionNode (selectedDirection=ZMinus toolParams=0.02, 0.02)
                      Until DISTANCE (allowActions=false deceleration=3 distanceNodeType=STOP) Distance=0.035; motionParameters(blendRadius=0)
                    MoveDirectionNode (selectedDirection=ZPlus toolParams=0.02, 0.02)
                      Until DISTANCE (allowActions=false deceleration=3 distanceNodeType=STOP) Distance=0.035; motionParameters(blendRadius=0)
              SuppressedNode
                Folder Buje17
                  Xfin := ((0.50165*Xp)-(Xd)-(-0.0127*(1/m2)))*(-1)
                  Yfin := ((-0.0127*Yp)-(Yd)+(0.50165*m1))*(-1)
                  rotaciones := get_actual_tcp_pose()
                  var_3 := rotaciones[3]
                  var_4 := rotaciones[4]
                  var_5 := rotaciones[5]
                  PosFinal := p[Xfin+0.00208915,Yfin+0.00208915,0.03,var_3,var_4,var_5]
                  MoveL speed 250 mm/s, acceleration 1200 mm/s^2 (useActiveTCP=true) feature=Base
                    MoveJ speed 60 deg/s, acceleration 80 deg/s^2 (useActiveTCP=true) feature=Base
                      Waypoint Waypoint (Variable): motionParameters(jointSpeed=1.047198 jointAcceleration=1.396263 cartesianSpeed=0.15 cartesianAcceleration=0.2); variable=PosFinal
                    MoveDirectionNode (selectedDirection=ZMinus toolParams=0.02, 0.02)
                      Until DISTANCE (allowActions=false deceleration=3 distanceNodeType=STOP) Distance=0.035; motionParameters(blendRadius=0)
                    MoveDirectionNode (selectedDirection=ZPlus toolParams=0.02, 0.02)
                      Until DISTANCE (allowActions=false deceleration=3 distanceNodeType=STOP) Distance=0.035; motionParameters(blendRadius=0)
              SuppressedNode
                Folder Buje18
                  Xfin := ((0.52705*Xp)-(Xd)-(-0.0127*(1/m2)))*(-1)
                  Yfin := ((-0.0127*Yp)-(Yd)+(0.52705*m1))*(-1)
                  rotaciones := get_actual_tcp_pose()
                  var_3 := rotaciones[3]
                  var_4 := rotaciones[4]
                  var_5 := rotaciones[5]
                  PosFinal := p[Xfin+0.00208915,Yfin+0.00208915,0.03,var_3,var_4,var_5]
                  MoveL speed 250 mm/s, acceleration 1200 mm/s^2 (useActiveTCP=true) feature=Base
                    MoveJ speed 60 deg/s, acceleration 80 deg/s^2 (useActiveTCP=true) feature=Base
                      Waypoint Waypoint (Variable): motionParameters(jointSpeed=1.047198 jointAcceleration=1.396263 cartesianSpeed=0.15 cartesianAcceleration=0.2); variable=PosFinal
                    MoveDirectionNode (selectedDirection=ZMinus toolParams=0.02, 0.02)
                      Until DISTANCE (allowActions=false deceleration=3 distanceNodeType=STOP) Distance=0.035; motionParameters(blendRadius=0)
                    MoveDirectionNode (selectedDirection=ZPlus toolParams=0.02, 0.02)
                      Until DISTANCE (allowActions=false deceleration=3 distanceNodeType=STOP) Distance=0.035; motionParameters(blendRadius=0)
              SuppressedNode
                Folder Buje19
                  Xfin := ((0.55245*Xp)-(Xd)-(-0.0127*(1/m2)))*(-1)
                  Yfin := ((-0.0127*Yp)-(Yd)+(0.55245*m1))*(-1)
                  rotaciones := get_actual_tcp_pose()
                  var_3 := rotaciones[3]
                  var_4 := rotaciones[4]
                  var_5 := rotaciones[5]
                  PosFinal := p[Xfin+0.00208915,Yfin+0.00208915,0.03,var_3,var_4,var_5]
                  MoveL speed 250 mm/s, acceleration 1200 mm/s^2 (useActiveTCP=true) feature=Base
                    MoveJ speed 60 deg/s, acceleration 80 deg/s^2 (useActiveTCP=true) feature=Base
                      Waypoint Waypoint (Variable): motionParameters(jointSpeed=1.047198 jointAcceleration=1.396263 cartesianSpeed=0.15 cartesianAcceleration=0.2); variable=PosFinal
                    MoveDirectionNode (selectedDirection=ZMinus toolParams=0.02, 0.02)
                      Until DISTANCE (allowActions=false deceleration=3 distanceNodeType=STOP) Distance=0.035; motionParameters(blendRadius=0)
                    MoveDirectionNode (selectedDirection=ZPlus toolParams=0.02, 0.02)
                      Until DISTANCE (allowActions=false deceleration=3 distanceNodeType=STOP) Distance=0.035; motionParameters(blendRadius=0)
              SuppressedNode
                Folder Buje20
                  Xfin := ((0.57785*Xp)-(Xd)-(-0.0127*(1/m2)))*(-1)
                  Yfin := ((-0.0127*Yp)-(Yd)+(0.57785*m1))*(-1)
                  rotaciones := get_actual_tcp_pose()
                  var_3 := rotaciones[3]
                  var_4 := rotaciones[4]
                  var_5 := rotaciones[5]
                  PosFinal := p[Xfin+0.00208915,Yfin+0.00208915,0.03,var_3,var_4,var_5]
                  MoveL speed 250 mm/s, acceleration 1200 mm/s^2 (useActiveTCP=true) feature=Base
                    MoveJ speed 60 deg/s, acceleration 80 deg/s^2 (useActiveTCP=true) feature=Base
                      Waypoint Waypoint (Variable): motionParameters(jointSpeed=1.047198 jointAcceleration=1.396263 cartesianSpeed=0.15 cartesianAcceleration=0.2); variable=PosFinal
                    MoveDirectionNode (selectedDirection=ZMinus toolParams=0.02, 0.02)
                      Until DISTANCE (allowActions=false deceleration=3 distanceNodeType=STOP) Distance=0.035; motionParameters(blendRadius=0)
                    MoveDirectionNode (selectedDirection=ZPlus toolParams=0.02, 0.02)
                      Until DISTANCE (allowActions=false deceleration=3 distanceNodeType=STOP) Distance=0.035; motionParameters(blendRadius=0)
              SuppressedNode
                Folder Buje21
                  Xfin := ((0.60325*Xp)-(Xd)-(-0.0127*(1/m2)))*(-1)
                  Yfin := ((-0.0127*Yp)-(Yd)+(0.60325*m1))*(-1)
                  rotaciones := get_actual_tcp_pose()
                  var_3 := rotaciones[3]
                  var_4 := rotaciones[4]
                  var_5 := rotaciones[5]
                  PosFinal := p[Xfin+0.00208915,Yfin+0.00208915,0.03,var_3,var_4,var_5]
                  MoveL speed 250 mm/s, acceleration 1200 mm/s^2 (useActiveTCP=true) feature=Base
                    MoveJ speed 60 deg/s, acceleration 80 deg/s^2 (useActiveTCP=true) feature=Base
                      Waypoint Waypoint (Variable): motionParameters(jointSpeed=1.047198 jointAcceleration=1.396263 cartesianSpeed=0.15 cartesianAcceleration=0.2); variable=PosFinal
                    MoveDirectionNode (selectedDirection=ZMinus toolParams=0.02, 0.02)
                      Until DISTANCE (allowActions=false deceleration=3 distanceNodeType=STOP) Distance=0.035; motionParameters(blendRadius=0)
                    MoveDirectionNode (selectedDirection=ZPlus toolParams=0.02, 0.02)
                      Until DISTANCE (allowActions=false deceleration=3 distanceNodeType=STOP) Distance=0.035; motionParameters(blendRadius=0)
              SuppressedNode
                Folder Buje22
                  Xfin := ((0.62865*Xp)-(Xd)-(-0.0127*(1/m2)))*(-1)
                  Yfin := ((-0.0127*Yp)-(Yd)+(0.62865*m1))*(-1)
                  rotaciones := get_actual_tcp_pose()
                  var_3 := rotaciones[3]
                  var_4 := rotaciones[4]
                  var_5 := rotaciones[5]
                  PosFinal := p[Xfin+0.00208915,Yfin+0.00208915,0.03,var_3,var_4,var_5]
                  MoveL speed 250 mm/s, acceleration 1200 mm/s^2 (useActiveTCP=true) feature=Base
                    MoveJ speed 60 deg/s, acceleration 80 deg/s^2 (useActiveTCP=true) feature=Base
                      Waypoint Waypoint (Variable): motionParameters(jointSpeed=1.047198 jointAcceleration=1.396263 cartesianSpeed=0.15 cartesianAcceleration=0.2); variable=PosFinal
                    MoveDirectionNode (selectedDirection=ZMinus toolParams=0.02, 0.02)
                      Until DISTANCE (allowActions=false deceleration=3 distanceNodeType=STOP) Distance=0.035; motionParameters(blendRadius=0)
                    MoveDirectionNode (selectedDirection=ZPlus toolParams=0.02, 0.02)
                      Until DISTANCE (allowActions=false deceleration=3 distanceNodeType=STOP) Distance=0.035; motionParameters(blendRadius=0)
              SuppressedNode
                Folder Buje23
                  Xfin := ((0.65405*Xp)-(Xd)-(-0.0127*(1/m2)))*(-1)
                  Yfin := ((-0.0127*Yp)-(Yd)+(0.65405*m1))*(-1)
                  rotaciones := get_actual_tcp_pose()
                  var_3 := rotaciones[3]
                  var_4 := rotaciones[4]
                  var_5 := rotaciones[5]
                  PosFinal := p[Xfin+0.00208915,Yfin+0.00208915,0.03,var_3,var_4,var_5]
                  MoveL speed 250 mm/s, acceleration 1200 mm/s^2 (useActiveTCP=true) feature=Base
                    MoveJ speed 60 deg/s, acceleration 80 deg/s^2 (useActiveTCP=true) feature=Base
                      Waypoint Waypoint (Variable): motionParameters(jointSpeed=1.047198 jointAcceleration=1.396263 cartesianSpeed=0.15 cartesianAcceleration=0.2); variable=PosFinal
                    MoveDirectionNode (selectedDirection=ZMinus toolParams=0.02, 0.02)
                      Until DISTANCE (allowActions=false deceleration=3 distanceNodeType=STOP) Distance=0.035; motionParameters(blendRadius=0)
                    MoveDirectionNode (selectedDirection=ZPlus toolParams=0.02, 0.02)
                      Until DISTANCE (allowActions=false deceleration=3 distanceNodeType=STOP) Distance=0.035; motionParameters(blendRadius=0)
              SuppressedNode
                Folder Buje24
                  Xfin := ((0.67945*Xp)-(Xd)-(-0.0127*(1/m2)))*(-1)
                  Yfin := ((-0.0127*Yp)-(Yd)+(0.67945*m1))*(-1)
                  rotaciones := get_actual_tcp_pose()
                  var_3 := rotaciones[3]
                  var_4 := rotaciones[4]
                  var_5 := rotaciones[5]
                  PosFinal := p[Xfin+0.00208915,Yfin+0.00208915,0.03,var_3,var_4,var_5]
                  MoveL speed 250 mm/s, acceleration 1200 mm/s^2 (useActiveTCP=true) feature=Base
                    MoveJ speed 60 deg/s, acceleration 80 deg/s^2 (useActiveTCP=true) feature=Base
                      Waypoint Waypoint (Variable): motionParameters(jointSpeed=1.047198 jointAcceleration=1.396263 cartesianSpeed=0.15 cartesianAcceleration=0.2); variable=PosFinal
                    MoveDirectionNode (selectedDirection=ZMinus toolParams=0.02, 0.02)
                      Until DISTANCE (allowActions=false deceleration=3 distanceNodeType=STOP) Distance=0.035; motionParameters(blendRadius=0)
                    MoveDirectionNode (selectedDirection=ZPlus toolParams=0.02, 0.02)
                      Until DISTANCE (allowActions=false deceleration=3 distanceNodeType=STOP) Distance=0.035; motionParameters(blendRadius=0)
              Folder Buje25
                Xfin := ((0.70485*Xp)-(Xd)-(-0.0127*(1/m2)))*(-1)
                Yfin := ((-0.0127*Yp)-(Yd)+(0.70485*m1))*(-1)
                rotaciones := get_actual_tcp_pose()
                var_3 := rotaciones[3]
                var_4 := rotaciones[4]
                var_5 := rotaciones[5]
                PosFinal := p[Xfin+0.00208915,Yfin+0.00208915,0.03,var_3,var_4,var_5]
                MoveL speed 250 mm/s, acceleration 1200 mm/s^2 (useActiveTCP=true) feature=Base
                  MoveJ speed 60 deg/s, acceleration 80 deg/s^2 (useActiveTCP=true) feature=Base
                    Waypoint Waypoint (Variable): motionParameters(jointSpeed=1.047198 jointAcceleration=1.396263 cartesianSpeed=0.15 cartesianAcceleration=0.2); variable=PosFinal
                  MoveDirectionNode (selectedDirection=ZMinus toolParams=0.02, 0.02)
                    Until DISTANCE (allowActions=false deceleration=3 distanceNodeType=STOP) Distance=0.035; motionParameters(blendRadius=0)
                  MoveDirectionNode (selectedDirection=ZPlus toolParams=0.02, 0.02)
                    Until DISTANCE (allowActions=false deceleration=3 distanceNodeType=STOP) Distance=0.035; motionParameters(blendRadius=0)
              Folder Buje26
                Xfin := ((0.73025*Xp)-(Xd)-(-0.0127*(1/m2)))*(-1)
                Yfin := ((-0.0127*Yp)-(Yd)+(0.73025*m1))*(-1)
                rotaciones := get_actual_tcp_pose()
                var_3 := rotaciones[3]
                var_4 := rotaciones[4]
                var_5 := rotaciones[5]
                PosFinal := p[Xfin+0.00208915,Yfin+0.00208915,0.03,var_3,var_4,var_5]
                MoveL speed 250 mm/s, acceleration 1200 mm/s^2 (useActiveTCP=true) feature=Base
                  MoveJ speed 60 deg/s, acceleration 80 deg/s^2 (useActiveTCP=true) feature=Base
                    Waypoint Waypoint (Variable): motionParameters(jointSpeed=1.047198 jointAcceleration=1.396263 cartesianSpeed=0.15 cartesianAcceleration=0.2); variable=PosFinal
                  MoveDirectionNode (selectedDirection=ZMinus toolParams=0.02, 0.02)
                    Until DISTANCE (allowActions=false deceleration=3 distanceNodeType=STOP) Distance=0.035; motionParameters(blendRadius=0)
                  MoveDirectionNode (selectedDirection=ZPlus toolParams=0.02, 0.02)
                    Until DISTANCE (allowActions=false deceleration=3 distanceNodeType=STOP) Distance=0.035; motionParameters(blendRadius=0)
              Folder Buje27
                Xfin := ((0.75565*Xp)-(Xd)-(-0.0127*(1/m2)))*(-1)
                Yfin := ((-0.0127*Yp)-(Yd)+(0.75565*m1))*(-1)
                rotaciones := get_actual_tcp_pose()
                var_3 := rotaciones[3]
                var_4 := rotaciones[4]
                var_5 := rotaciones[5]
                PosFinal := p[Xfin+0.00208915,Yfin+0.00208915,0.03,var_3,var_4,var_5]
                MoveL speed 250 mm/s, acceleration 1200 mm/s^2 (useActiveTCP=true) feature=Base
                  MoveJ speed 60 deg/s, acceleration 80 deg/s^2 (useActiveTCP=true) feature=Base
                    Waypoint Waypoint (Variable): motionParameters(jointSpeed=1.047198 jointAcceleration=1.396263 cartesianSpeed=0.15 cartesianAcceleration=0.2); variable=PosFinal
                  MoveDirectionNode (selectedDirection=ZMinus toolParams=0.02, 0.02)
                    Until DISTANCE (allowActions=false deceleration=3 distanceNodeType=STOP) Distance=0.035; motionParameters(blendRadius=0)
                  MoveDirectionNode (selectedDirection=ZPlus toolParams=0.02, 0.02)
                    Until DISTANCE (allowActions=false deceleration=3 distanceNodeType=STOP) Distance=0.035; motionParameters(blendRadius=0)
              Popup Message (haltProgram=false message=oi inputType=Text)
            MoveJ speed 60 deg/s, acceleration 80 deg/s^2 (useActiveTCP=true) feature=Base
              Waypoint Casa1: TCP in base x=-397.714 y=-209.387 z=130.553 mm, rx=2.0075 ry=-2.3998 rz=-0.0199 rad; joints [8.28, -111.842, 141.427, -30.137, 99.306, -0.058] deg; TCP offset x=0.411 y=-218.298 z=37.994 mm, rx=1.558 ry=-0.1255 rz=0.1212 rad
            Folder Buje1
              Xfin := ((0.09525*Xp)-(Xd)-(0.3937*(1/m2)))*(-1)
              Yfin := ((0.3937*Yp)-(Yd)+(0.09525*m1))*(-1)
              rotaciones := get_actual_tcp_pose()
              var_3 := rotaciones[3]
              var_4 := rotaciones[4]
              var_5 := rotaciones[5]
              PosFinal := p[Xfin+0.00208915,Yfin+0.00208915,-0.44,var_3,var_4,var_5]
              MoveL speed 250 mm/s, acceleration 1200 mm/s^2 (useActiveTCP=true) feature=Base
                MoveJ speed 60 deg/s, acceleration 80 deg/s^2 (useActiveTCP=true) feature=Base
                  Waypoint Waypoint (Variable): motionParameters(jointSpeed=1.047198 jointAcceleration=1.396263 cartesianSpeed=0.15 cartesianAcceleration=0.2); variable=PosFinal
                MoveDirectionNode (selectedDirection=ZMinus toolParams=0.02, 0.02)
                  Until DISTANCE (allowActions=false deceleration=3 distanceNodeType=STOP) Distance=0.075; motionParameters(blendRadius=0)
                MoveDirectionNode (selectedDirection=ZPlus toolParams=0.02, 0.02)
                  Until DISTANCE (allowActions=false deceleration=3 distanceNodeType=STOP) Distance=0.075; motionParameters(blendRadius=0)
            Folder Buje2
              Xfin := ((0.12065*Xp)-(Xd)-(0.3937*(1/m2)))*(-1)
              Yfin := ((0.3937*Yp)-(Yd)+(0.12065*m1))*(-1)
              rotaciones := get_actual_tcp_pose()
              var_3 := rotaciones[3]
              var_4 := rotaciones[4]
              var_5 := rotaciones[5]
              PosFinal := p[Xfin+0.00208915,Yfin+0.00208915,-0.44,var_3,var_4,var_5]
              MoveL speed 250 mm/s, acceleration 1200 mm/s^2 (useActiveTCP=true) feature=Base
                MoveJ speed 60 deg/s, acceleration 80 deg/s^2 (useActiveTCP=true) feature=Base
                  Waypoint Waypoint (Variable): motionParameters(jointSpeed=1.047198 jointAcceleration=1.396263 cartesianSpeed=0.15 cartesianAcceleration=0.2); variable=PosFinal
                MoveDirectionNode (selectedDirection=ZMinus toolParams=0.02, 0.02)
                  Until DISTANCE (allowActions=false deceleration=3 distanceNodeType=STOP) Distance=0.075; motionParameters(blendRadius=0)
                MoveDirectionNode (selectedDirection=ZPlus toolParams=0.02, 0.02)
                  Until DISTANCE (allowActions=false deceleration=3 distanceNodeType=STOP) Distance=0.075; motionParameters(blendRadius=0)
            Folder Buje3
              Xfin := ((0.14605*Xp)-(Xd)-(0.3937*(1/m2)))*(-1)
              Yfin := ((0.3937*Yp)-(Yd)+(0.14605*m1))*(-1)
              rotaciones := get_actual_tcp_pose()
              var_3 := rotaciones[3]
              var_4 := rotaciones[4]
              var_5 := rotaciones[5]
              PosFinal := p[Xfin+0.00208915,Yfin+0.00208915,-0.440,var_3,var_4,var_5]
              MoveL speed 250 mm/s, acceleration 1200 mm/s^2 (useActiveTCP=true) feature=Base
                MoveJ speed 60 deg/s, acceleration 80 deg/s^2 (useActiveTCP=true) feature=Base
                  Waypoint Waypoint (Variable): motionParameters(jointSpeed=1.047198 jointAcceleration=1.396263 cartesianSpeed=0.15 cartesianAcceleration=0.2); variable=PosFinal
                MoveDirectionNode (selectedDirection=ZMinus toolParams=0.02, 0.02)
                  Until DISTANCE (allowActions=false deceleration=3 distanceNodeType=STOP) Distance=0.075; motionParameters(blendRadius=0)
                MoveDirectionNode (selectedDirection=ZPlus toolParams=0.02, 0.02)
                  Until DISTANCE (allowActions=false deceleration=3 distanceNodeType=STOP) Distance=0.075; motionParameters(blendRadius=0)
            Folder Buje4
              Xfin := ((0.17145*Xp)-(Xd)-(0.3937*(1/m2)))*(-1)
              Yfin := ((0.3937*Yp)-(Yd)+(0.17145*m1))*(-1)
              rotaciones := get_actual_tcp_pose()
              var_3 := rotaciones[3]
              var_4 := rotaciones[4]
              var_5 := rotaciones[5]
              PosFinal := p[Xfin+0.00208915,Yfin+0.00208915,-0.44,var_3,var_4,var_5]
              MoveL speed 250 mm/s, acceleration 1200 mm/s^2 (useActiveTCP=true) feature=Base
                MoveJ speed 60 deg/s, acceleration 80 deg/s^2 (useActiveTCP=true) feature=Base
                  Waypoint Waypoint (Variable): motionParameters(jointSpeed=1.047198 jointAcceleration=1.396263 cartesianSpeed=0.15 cartesianAcceleration=0.2); variable=PosFinal
                MoveDirectionNode (selectedDirection=ZMinus toolParams=0.02, 0.02)
                  Until DISTANCE (allowActions=false deceleration=3 distanceNodeType=STOP) Distance=0.075; motionParameters(blendRadius=0)
                MoveDirectionNode (selectedDirection=ZPlus toolParams=0.02, 0.02)
                  Until DISTANCE (allowActions=false deceleration=3 distanceNodeType=STOP) Distance=0.075; motionParameters(blendRadius=0)
            Folder Buje5
              Xfin := ((0.19685*Xp)-(Xd)-(0.3937*(1/m2)))*(-1)
              Yfin := ((0.3937*Yp)-(Yd)+(0.19685*m1))*(-1)
              rotaciones := get_actual_tcp_pose()
              var_3 := rotaciones[3]
              var_4 := rotaciones[4]
              var_5 := rotaciones[5]
              PosFinal := p[Xfin+0.00208915,Yfin+0.00208915,-0.44,var_3,var_4,var_5]
              MoveL speed 250 mm/s, acceleration 1200 mm/s^2 (useActiveTCP=true) feature=Base
                MoveJ speed 60 deg/s, acceleration 80 deg/s^2 (useActiveTCP=true) feature=Base
                  Waypoint Waypoint (Variable): motionParameters(jointSpeed=1.047198 jointAcceleration=1.396263 cartesianSpeed=0.15 cartesianAcceleration=0.2); variable=PosFinal
                MoveDirectionNode (selectedDirection=ZMinus toolParams=0.02, 0.02)
                  Until DISTANCE (allowActions=false deceleration=3 distanceNodeType=STOP) Distance=0.075; motionParameters(blendRadius=0)
                MoveDirectionNode (selectedDirection=ZPlus toolParams=0.02, 0.02)
                  Until DISTANCE (allowActions=false deceleration=3 distanceNodeType=STOP) Distance=0.075; motionParameters(blendRadius=0)
            Folder Buje6
              Xfin := ((0.22225*Xp)-(Xd)-(0.3937*(1/m2)))*(-1)
              Yfin := ((0.3937*Yp)-(Yd)+(0.22225*m1))*(-1)
              rotaciones := get_actual_tcp_pose()
              var_3 := rotaciones[3]
              var_4 := rotaciones[4]
              var_5 := rotaciones[5]
              PosFinal := p[Xfin+0.00208915,Yfin+0.00208915,-0.44,var_3,var_4,var_5]
              MoveL speed 250 mm/s, acceleration 1200 mm/s^2 (useActiveTCP=true) feature=Base
                MoveJ speed 60 deg/s, acceleration 80 deg/s^2 (useActiveTCP=true) feature=Base
                  Waypoint Waypoint (Variable): motionParameters(jointSpeed=1.047198 jointAcceleration=1.396263 cartesianSpeed=0.15 cartesianAcceleration=0.2); variable=PosFinal
                MoveDirectionNode (selectedDirection=ZMinus toolParams=0.02, 0.02)
                  Until DISTANCE (allowActions=false deceleration=3 distanceNodeType=STOP) Distance=0.075; motionParameters(blendRadius=0)
                MoveDirectionNode (selectedDirection=ZPlus toolParams=0.02, 0.02)
                  Until DISTANCE (allowActions=false deceleration=3 distanceNodeType=STOP) Distance=0.075; motionParameters(blendRadius=0)
            Folder Buje7
              Xfin := ((0.24765*Xp)-(Xd)-(0.3937*(1/m2)))*(-1)
              Yfin := ((0.3937*Yp)-(Yd)+(0.24765*m1))*(-1)
              rotaciones := get_actual_tcp_pose()
              var_3 := rotaciones[3]
              var_4 := rotaciones[4]
              var_5 := rotaciones[5]
              PosFinal := p[Xfin+0.00208915,Yfin+0.00208915,-0.44,var_3,var_4,var_5]
              MoveL speed 250 mm/s, acceleration 1200 mm/s^2 (useActiveTCP=true) feature=Base
                MoveJ speed 60 deg/s, acceleration 80 deg/s^2 (useActiveTCP=true) feature=Base
                  Waypoint Waypoint (Variable): motionParameters(jointSpeed=1.047198 jointAcceleration=1.396263 cartesianSpeed=0.15 cartesianAcceleration=0.2); variable=PosFinal
                MoveDirectionNode (selectedDirection=ZMinus toolParams=0.02, 0.02)
                  Until DISTANCE (allowActions=false deceleration=3 distanceNodeType=STOP) Distance=0.075; motionParameters(blendRadius=0)
                MoveDirectionNode (selectedDirection=ZPlus toolParams=0.02, 0.02)
                  Until DISTANCE (allowActions=false deceleration=3 distanceNodeType=STOP) Distance=0.075; motionParameters(blendRadius=0)
            Folder Buje8
              Xfin := ((0.27305*Xp)-(Xd)-(0.3937*(1/m2)))*(-1)
              Yfin := ((0.3937*Yp)-(Yd)+(0.27305*m1))*(-1)
              rotaciones := get_actual_tcp_pose()
              var_3 := rotaciones[3]
              var_4 := rotaciones[4]
              var_5 := rotaciones[5]
              PosFinal := p[Xfin+0.00208915,Yfin+0.00208915,-0.44,var_3,var_4,var_5]
              MoveL speed 250 mm/s, acceleration 1200 mm/s^2 (useActiveTCP=true) feature=Base
                MoveJ speed 60 deg/s, acceleration 80 deg/s^2 (useActiveTCP=true) feature=Base
                  Waypoint Waypoint (Variable): motionParameters(jointSpeed=1.047198 jointAcceleration=1.396263 cartesianSpeed=0.15 cartesianAcceleration=0.2); variable=PosFinal
                MoveDirectionNode (selectedDirection=ZMinus toolParams=0.02, 0.02)
                  Until DISTANCE (allowActions=false deceleration=3 distanceNodeType=STOP) Distance=0.075; motionParameters(blendRadius=0)
                MoveDirectionNode (selectedDirection=ZPlus toolParams=0.02, 0.02)
                  Until DISTANCE (allowActions=false deceleration=3 distanceNodeType=STOP) Distance=0.075; motionParameters(blendRadius=0)
            Folder Buje9
              Xfin := ((0.29845*Xp)-(Xd)-(0.3937*(1/m2)))*(-1)
              Yfin := ((0.3937*Yp)-(Yd)+(0.29845*m1))*(-1)
              rotaciones := get_actual_tcp_pose()
              var_3 := rotaciones[3]
              var_4 := rotaciones[4]
              var_5 := rotaciones[5]
              PosFinal := p[Xfin+0.00208915,Yfin+0.00208915,-0.44,var_3,var_4,var_5]
              MoveL speed 250 mm/s, acceleration 1200 mm/s^2 (useActiveTCP=true) feature=Base
                MoveJ speed 60 deg/s, acceleration 80 deg/s^2 (useActiveTCP=true) feature=Base
                  Waypoint Waypoint (Variable): motionParameters(jointSpeed=1.047198 jointAcceleration=1.396263 cartesianSpeed=0.15 cartesianAcceleration=0.2); variable=PosFinal
                MoveDirectionNode (selectedDirection=ZMinus toolParams=0.02, 0.02)
                  Until DISTANCE (allowActions=false deceleration=3 distanceNodeType=STOP) Distance=0.075; motionParameters(blendRadius=0)
                MoveDirectionNode (selectedDirection=ZPlus toolParams=0.02, 0.02)
                  Until DISTANCE (allowActions=false deceleration=3 distanceNodeType=STOP) Distance=0.075; motionParameters(blendRadius=0)
            Folder Buje10
              Xfin := ((0.32385*Xp)-(Xd)-(0.3937*(1/m2)))*(-1)
              Yfin := ((0.3937*Yp)-(Yd)+(0.32385*m1))*(-1)
              rotaciones := get_actual_tcp_pose()
              var_3 := rotaciones[3]
              var_4 := rotaciones[4]
              var_5 := rotaciones[5]
              PosFinal := p[Xfin+0.00208915,Yfin+0.00208915,-0.44,var_3,var_4,var_5]
              MoveL speed 250 mm/s, acceleration 1200 mm/s^2 (useActiveTCP=true) feature=Base
                MoveJ speed 60 deg/s, acceleration 80 deg/s^2 (useActiveTCP=true) feature=Base
                  Waypoint Waypoint (Variable): motionParameters(jointSpeed=1.047198 jointAcceleration=1.396263 cartesianSpeed=0.15 cartesianAcceleration=0.2); variable=PosFinal
                MoveDirectionNode (selectedDirection=ZMinus toolParams=0.02, 0.02)
                  Until DISTANCE (allowActions=false deceleration=3 distanceNodeType=STOP) Distance=0.075; motionParameters(blendRadius=0)
                MoveDirectionNode (selectedDirection=ZPlus toolParams=0.02, 0.02)
                  Until DISTANCE (allowActions=false deceleration=3 distanceNodeType=STOP) Distance=0.075; motionParameters(blendRadius=0)
            Folder Buje11
              Xfin := ((0.34925*Xp)-(Xd)-(0.3937*(1/m2)))*(-1)
              Yfin := ((0.3937*Yp)-(Yd)+(0.34925*m1))*(-1)
              rotaciones := get_actual_tcp_pose()
              var_3 := rotaciones[3]
              var_4 := rotaciones[4]
              var_5 := rotaciones[5]
              PosFinal := p[Xfin+0.00208915,Yfin+0.00208915,-0.44,var_3,var_4,var_5]
              MoveL speed 250 mm/s, acceleration 1200 mm/s^2 (useActiveTCP=true) feature=Base
                MoveJ speed 60 deg/s, acceleration 80 deg/s^2 (useActiveTCP=true) feature=Base
                  Waypoint Waypoint (Variable): motionParameters(jointSpeed=1.047198 jointAcceleration=1.396263 cartesianSpeed=0.15 cartesianAcceleration=0.2); variable=PosFinal
                MoveDirectionNode (selectedDirection=ZMinus toolParams=0.02, 0.02)
                  Until DISTANCE (allowActions=false deceleration=3 distanceNodeType=STOP) Distance=0.075; motionParameters(blendRadius=0)
                MoveDirectionNode (selectedDirection=ZPlus toolParams=0.02, 0.02)
                  Until DISTANCE (allowActions=false deceleration=3 distanceNodeType=STOP) Distance=0.075; motionParameters(blendRadius=0)
            Folder Buje12
              Xfin := ((0.37465*Xp)-(Xd)-(0.3937*(1/m2)))*(-1)
              Yfin := ((0.3937*Yp)-(Yd)+(0.37465*m1))*(-1)
              rotaciones := get_actual_tcp_pose()
              var_3 := rotaciones[3]
              var_4 := rotaciones[4]
              var_5 := rotaciones[5]
              PosFinal := p[Xfin+0.00208915,Yfin+0.00208915,-0.44,var_3,var_4,var_5]
              MoveL speed 250 mm/s, acceleration 1200 mm/s^2 (useActiveTCP=true) feature=Base
                MoveJ speed 60 deg/s, acceleration 80 deg/s^2 (useActiveTCP=true) feature=Base
                  Waypoint Waypoint (Variable): motionParameters(jointSpeed=1.047198 jointAcceleration=1.396263 cartesianSpeed=0.15 cartesianAcceleration=0.2); variable=PosFinal
                MoveDirectionNode (selectedDirection=ZMinus toolParams=0.02, 0.02)
                  Until DISTANCE (allowActions=false deceleration=3 distanceNodeType=STOP) Distance=0.075; motionParameters(blendRadius=0)
                MoveDirectionNode (selectedDirection=ZPlus toolParams=0.02, 0.02)
                  Until DISTANCE (allowActions=false deceleration=3 distanceNodeType=STOP) Distance=0.075; motionParameters(blendRadius=0)
            Folder Buje13
              Xfin := ((0.40005*Xp)-(Xd)-(0.3937*(1/m2)))*(-1)
              Yfin := ((0.3937*Yp)-(Yd)+(0.40005*m1))*(-1)
              rotaciones := get_actual_tcp_pose()
              var_3 := rotaciones[3]
              var_4 := rotaciones[4]
              var_5 := rotaciones[5]
              PosFinal := p[Xfin+0.00208915,Yfin+0.00208915,-0.44,var_3,var_4,var_5]
              MoveL speed 250 mm/s, acceleration 1200 mm/s^2 (useActiveTCP=true) feature=Base
                MoveJ speed 60 deg/s, acceleration 80 deg/s^2 (useActiveTCP=true) feature=Base
                  Waypoint Waypoint (Variable): motionParameters(jointSpeed=1.047198 jointAcceleration=1.396263 cartesianSpeed=0.15 cartesianAcceleration=0.2); variable=PosFinal
                MoveDirectionNode (selectedDirection=ZMinus toolParams=0.02, 0.02)
                  Until DISTANCE (allowActions=false deceleration=3 distanceNodeType=STOP) Distance=0.075; motionParameters(blendRadius=0)
                MoveDirectionNode (selectedDirection=ZPlus toolParams=0.02, 0.02)
                  Until DISTANCE (allowActions=false deceleration=3 distanceNodeType=STOP) Distance=0.075; motionParameters(blendRadius=0)
            Folder Buje14
              Xfin := ((0.42545*Xp)-(Xd)-(0.3937*(1/m2)))*(-1)
              Yfin := ((0.3937*Yp)-(Yd)+(0.42545*m1))*(-1)
              rotaciones := get_actual_tcp_pose()
              var_3 := rotaciones[3]
              var_4 := rotaciones[4]
              var_5 := rotaciones[5]
              PosFinal := p[Xfin+0.00208915,Yfin+0.00208915,-0.44,var_3,var_4,var_5]
              MoveL speed 250 mm/s, acceleration 1200 mm/s^2 (useActiveTCP=true) feature=Base
                MoveJ speed 60 deg/s, acceleration 80 deg/s^2 (useActiveTCP=true) feature=Base
                  Waypoint Waypoint (Variable): motionParameters(jointSpeed=1.047198 jointAcceleration=1.396263 cartesianSpeed=0.15 cartesianAcceleration=0.2); variable=PosFinal
                MoveDirectionNode (selectedDirection=ZMinus toolParams=0.02, 0.02)
                  Until DISTANCE (allowActions=false deceleration=3 distanceNodeType=STOP) Distance=0.075; motionParameters(blendRadius=0)
                MoveDirectionNode (selectedDirection=ZPlus toolParams=0.02, 0.02)
                  Until DISTANCE (allowActions=false deceleration=3 distanceNodeType=STOP) Distance=0.075; motionParameters(blendRadius=0)
            Folder Buje15
              Xfin := ((0.45085*Xp)-(Xd)-(0.3937*(1/m2)))*(-1)
              Yfin := ((0.3937*Yp)-(Yd)+(0.45085*m1))*(-1)
              rotaciones := get_actual_tcp_pose()
              var_3 := rotaciones[3]
              var_4 := rotaciones[4]
              var_5 := rotaciones[5]
              PosFinal := p[Xfin+0.00208915,Yfin+0.00208915,-0.44,var_3,var_4,var_5]
              MoveL speed 250 mm/s, acceleration 1200 mm/s^2 (useActiveTCP=true) feature=Base
                MoveJ speed 60 deg/s, acceleration 80 deg/s^2 (useActiveTCP=true) feature=Base
                  Waypoint Waypoint (Variable): motionParameters(jointSpeed=1.047198 jointAcceleration=1.396263 cartesianSpeed=0.15 cartesianAcceleration=0.2); variable=PosFinal
                MoveDirectionNode (selectedDirection=ZMinus toolParams=0.02, 0.02)
                  Until DISTANCE (allowActions=false deceleration=3 distanceNodeType=STOP) Distance=0.075; motionParameters(blendRadius=0)
                MoveDirectionNode (selectedDirection=ZPlus toolParams=0.02, 0.02)
                  Until DISTANCE (allowActions=false deceleration=3 distanceNodeType=STOP) Distance=0.075; motionParameters(blendRadius=0)
            Folder Buje16
              Xfin := ((0.47625*Xp)-(Xd)-(0.3937*(1/m2)))*(-1)
              Yfin := ((0.3937*Yp)-(Yd)+(0.47625*m1))*(-1)
              rotaciones := get_actual_tcp_pose()
              var_3 := rotaciones[3]
              var_4 := rotaciones[4]
              var_5 := rotaciones[5]
              PosFinal := p[Xfin+0.00208915,Yfin+0.00208915,-0.44,var_3,var_4,var_5]
              MoveL speed 250 mm/s, acceleration 1200 mm/s^2 (useActiveTCP=true) feature=Base
                MoveJ speed 60 deg/s, acceleration 80 deg/s^2 (useActiveTCP=true) feature=Base
                  Waypoint Waypoint (Variable): motionParameters(jointSpeed=1.047198 jointAcceleration=1.396263 cartesianSpeed=0.15 cartesianAcceleration=0.2); variable=PosFinal
                MoveDirectionNode (selectedDirection=ZMinus toolParams=0.02, 0.02)
                  Until DISTANCE (allowActions=false deceleration=3 distanceNodeType=STOP) Distance=0.075; motionParameters(blendRadius=0)
                MoveDirectionNode (selectedDirection=ZPlus toolParams=0.02, 0.02)
                  Until DISTANCE (allowActions=false deceleration=3 distanceNodeType=STOP) Distance=0.075; motionParameters(blendRadius=0)
            Folder Buje17
              Xfin := ((0.50165*Xp)-(Xd)-(0.3937*(1/m2)))*(-1)
              Yfin := ((0.3937*Yp)-(Yd)+(0.50165*m1))*(-1)
              rotaciones := get_actual_tcp_pose()
              var_3 := rotaciones[3]
              var_4 := rotaciones[4]
              var_5 := rotaciones[5]
              PosFinal := p[Xfin+0.00208915,Yfin+0.00208915,-0.44,var_3,var_4,var_5]
              MoveL speed 250 mm/s, acceleration 1200 mm/s^2 (useActiveTCP=true) feature=Base
                MoveJ speed 60 deg/s, acceleration 80 deg/s^2 (useActiveTCP=true) feature=Base
                  Waypoint Waypoint (Variable): motionParameters(jointSpeed=1.047198 jointAcceleration=1.396263 cartesianSpeed=0.15 cartesianAcceleration=0.2); variable=PosFinal
                MoveDirectionNode (selectedDirection=ZMinus toolParams=0.02, 0.02)
                  Until DISTANCE (allowActions=false deceleration=3 distanceNodeType=STOP) Distance=0.075; motionParameters(blendRadius=0)
                MoveDirectionNode (selectedDirection=ZPlus toolParams=0.02, 0.02)
                  Until DISTANCE (allowActions=false deceleration=3 distanceNodeType=STOP) Distance=0.075; motionParameters(blendRadius=0)
            Folder Buje18
              Xfin := ((0.52705*Xp)-(Xd)-(0.3937*(1/m2)))*(-1)
              Yfin := ((0.3937*Yp)-(Yd)+(0.52705*m1))*(-1)
              rotaciones := get_actual_tcp_pose()
              var_3 := rotaciones[3]
              var_4 := rotaciones[4]
              var_5 := rotaciones[5]
              PosFinal := p[Xfin+0.00208915,Yfin+0.00208915,-0.44,var_3,var_4,var_5]
              MoveL speed 250 mm/s, acceleration 1200 mm/s^2 (useActiveTCP=true) feature=Base
                MoveJ speed 60 deg/s, acceleration 80 deg/s^2 (useActiveTCP=true) feature=Base
                  Waypoint Waypoint (Variable): motionParameters(jointSpeed=1.047198 jointAcceleration=1.396263 cartesianSpeed=0.15 cartesianAcceleration=0.2); variable=PosFinal
                MoveDirectionNode (selectedDirection=ZMinus toolParams=0.02, 0.02)
                  Until DISTANCE (allowActions=false deceleration=3 distanceNodeType=STOP) Distance=0.075; motionParameters(blendRadius=0)
                MoveDirectionNode (selectedDirection=ZPlus toolParams=0.02, 0.02)
                  Until DISTANCE (allowActions=false deceleration=3 distanceNodeType=STOP) Distance=0.075; motionParameters(blendRadius=0)
            Folder Buje19
              Xfin := ((0.55245*Xp)-(Xd)-(0.3937*(1/m2)))*(-1)
              Yfin := ((0.3937*Yp)-(Yd)+(0.55245*m1))*(-1)
              rotaciones := get_actual_tcp_pose()
              var_3 := rotaciones[3]
              var_4 := rotaciones[4]
              var_5 := rotaciones[5]
              PosFinal := p[Xfin+0.00208915,Yfin+0.00208915,-0.44,var_3,var_4,var_5]
              MoveL speed 250 mm/s, acceleration 1200 mm/s^2 (useActiveTCP=true) feature=Base
                MoveJ speed 60 deg/s, acceleration 80 deg/s^2 (useActiveTCP=true) feature=Base
                  Waypoint Waypoint (Variable): motionParameters(jointSpeed=1.047198 jointAcceleration=1.396263 cartesianSpeed=0.15 cartesianAcceleration=0.2); variable=PosFinal
                MoveDirectionNode (selectedDirection=ZMinus toolParams=0.02, 0.02)
                  Until DISTANCE (allowActions=false deceleration=3 distanceNodeType=STOP) Distance=0.075; motionParameters(blendRadius=0)
                MoveDirectionNode (selectedDirection=ZPlus toolParams=0.02, 0.02)
                  Until DISTANCE (allowActions=false deceleration=3 distanceNodeType=STOP) Distance=0.075; motionParameters(blendRadius=0)
            Folder Buje20
              Xfin := ((0.57785*Xp)-(Xd)-(0.3937*(1/m2)))*(-1)
              Yfin := ((0.3937*Yp)-(Yd)+(0.57785*m1))*(-1)
              rotaciones := get_actual_tcp_pose()
              var_3 := rotaciones[3]
              var_4 := rotaciones[4]
              var_5 := rotaciones[5]
              PosFinal := p[Xfin+0.00208915,Yfin+0.00208915,-0.44,var_3,var_4,var_5]
              MoveL speed 250 mm/s, acceleration 1200 mm/s^2 (useActiveTCP=true) feature=Base
                MoveJ speed 60 deg/s, acceleration 80 deg/s^2 (useActiveTCP=true) feature=Base
                  Waypoint Waypoint (Variable): motionParameters(jointSpeed=1.047198 jointAcceleration=1.396263 cartesianSpeed=0.15 cartesianAcceleration=0.2); variable=PosFinal
                MoveDirectionNode (selectedDirection=ZMinus toolParams=0.02, 0.02)
                  Until DISTANCE (allowActions=false deceleration=3 distanceNodeType=STOP) Distance=0.075; motionParameters(blendRadius=0)
                MoveDirectionNode (selectedDirection=ZPlus toolParams=0.02, 0.02)
                  Until DISTANCE (allowActions=false deceleration=3 distanceNodeType=STOP) Distance=0.075; motionParameters(blendRadius=0)
            Folder Buje21
              Xfin := ((0.60325*Xp)-(Xd)-(0.3937*(1/m2)))*(-1)
              Yfin := ((0.3937*Yp)-(Yd)+(0.60325*m1))*(-1)
              rotaciones := get_actual_tcp_pose()
              var_3 := rotaciones[3]
              var_4 := rotaciones[4]
              var_5 := rotaciones[5]
              PosFinal := p[Xfin+0.00208915,Yfin+0.00208915,-0.44,var_3,var_4,var_5]
              MoveL speed 250 mm/s, acceleration 1200 mm/s^2 (useActiveTCP=true) feature=Base
                MoveJ speed 60 deg/s, acceleration 80 deg/s^2 (useActiveTCP=true) feature=Base
                  Waypoint Waypoint (Variable): motionParameters(jointSpeed=1.047198 jointAcceleration=1.396263 cartesianSpeed=0.15 cartesianAcceleration=0.2); variable=PosFinal
                MoveDirectionNode (selectedDirection=ZMinus toolParams=0.02, 0.02)
                  Until DISTANCE (allowActions=false deceleration=3 distanceNodeType=STOP) Distance=0.075; motionParameters(blendRadius=0)
                MoveDirectionNode (selectedDirection=ZPlus toolParams=0.02, 0.02)
                  Until DISTANCE (allowActions=false deceleration=3 distanceNodeType=STOP) Distance=0.075; motionParameters(blendRadius=0)
            Folder Buje22
              Xfin := ((0.62865*Xp)-(Xd)-(0.3937*(1/m2)))*(-1)
              Yfin := ((0.3937*Yp)-(Yd)+(0.62865*m1))*(-1)
              rotaciones := get_actual_tcp_pose()
              var_3 := rotaciones[3]
              var_4 := rotaciones[4]
              var_5 := rotaciones[5]
              PosFinal := p[Xfin+0.00208915,Yfin+0.00208915,-0.44,var_3,var_4,var_5]
              MoveL speed 250 mm/s, acceleration 1200 mm/s^2 (useActiveTCP=true) feature=Base
                MoveJ speed 60 deg/s, acceleration 80 deg/s^2 (useActiveTCP=true) feature=Base
                  Waypoint Waypoint (Variable): motionParameters(jointSpeed=1.047198 jointAcceleration=1.396263 cartesianSpeed=0.15 cartesianAcceleration=0.2); variable=PosFinal
                MoveDirectionNode (selectedDirection=ZMinus toolParams=0.02, 0.02)
                  Until DISTANCE (allowActions=false deceleration=3 distanceNodeType=STOP) Distance=0.075; motionParameters(blendRadius=0)
                MoveDirectionNode (selectedDirection=ZPlus toolParams=0.02, 0.02)
                  Until DISTANCE (allowActions=false deceleration=3 distanceNodeType=STOP) Distance=0.075; motionParameters(blendRadius=0)
            Folder Buje23
              Xfin := ((0.65405*Xp)-(Xd)-(0.3937*(1/m2)))*(-1)
              Yfin := ((0.3937*Yp)-(Yd)+(0.65405*m1))*(-1)
              rotaciones := get_actual_tcp_pose()
              var_3 := rotaciones[3]
              var_4 := rotaciones[4]
              var_5 := rotaciones[5]
              PosFinal := p[Xfin+0.00208915,Yfin+0.00208915,-0.44,var_3,var_4,var_5]
              MoveL speed 250 mm/s, acceleration 1200 mm/s^2 (useActiveTCP=true) feature=Base
                MoveJ speed 60 deg/s, acceleration 80 deg/s^2 (useActiveTCP=true) feature=Base
                  Waypoint Waypoint (Variable): motionParameters(jointSpeed=1.047198 jointAcceleration=1.396263 cartesianSpeed=0.15 cartesianAcceleration=0.2); variable=PosFinal
                MoveDirectionNode (selectedDirection=ZMinus toolParams=0.02, 0.02)
                  Until DISTANCE (allowActions=false deceleration=3 distanceNodeType=STOP) Distance=0.075; motionParameters(blendRadius=0)
                MoveDirectionNode (selectedDirection=ZPlus toolParams=0.02, 0.02)
                  Until DISTANCE (allowActions=false deceleration=3 distanceNodeType=STOP) Distance=0.075; motionParameters(blendRadius=0)
            Folder Buje24
              Xfin := ((0.67945*Xp)-(Xd)-(0.3937*(1/m2)))*(-1)
              Yfin := ((0.3937*Yp)-(Yd)+(0.67945*m1))*(-1)
              rotaciones := get_actual_tcp_pose()
              var_3 := rotaciones[3]
              var_4 := rotaciones[4]
              var_5 := rotaciones[5]
              PosFinal := p[Xfin+0.00208915,Yfin+0.00208915,-0.44,var_3,var_4,var_5]
              MoveL speed 250 mm/s, acceleration 1200 mm/s^2 (useActiveTCP=true) feature=Base
                MoveJ speed 60 deg/s, acceleration 80 deg/s^2 (useActiveTCP=true) feature=Base
                  Waypoint Waypoint (Variable): motionParameters(jointSpeed=1.047198 jointAcceleration=1.396263 cartesianSpeed=0.15 cartesianAcceleration=0.2); variable=PosFinal
                MoveDirectionNode (selectedDirection=ZMinus toolParams=0.02, 0.02)
                  Until DISTANCE (allowActions=false deceleration=3 distanceNodeType=STOP) Distance=0.075; motionParameters(blendRadius=0)
                MoveDirectionNode (selectedDirection=ZPlus toolParams=0.02, 0.02)
                  Until DISTANCE (allowActions=false deceleration=3 distanceNodeType=STOP) Distance=0.075; motionParameters(blendRadius=0)
            Folder Buje25
              Xfin := ((0.70485*Xp)-(Xd)-(0.3937*(1/m2)))*(-1)
              Yfin := ((0.3937*Yp)-(Yd)+(0.70485*m1))*(-1)
              rotaciones := get_actual_tcp_pose()
              var_3 := rotaciones[3]
              var_4 := rotaciones[4]
              var_5 := rotaciones[5]
              PosFinal := p[Xfin+0.00208915,Yfin+0.00208915,-0.44,var_3,var_4,var_5]
              MoveL speed 250 mm/s, acceleration 1200 mm/s^2 (useActiveTCP=true) feature=Base
                MoveJ speed 60 deg/s, acceleration 80 deg/s^2 (useActiveTCP=true) feature=Base
                  Waypoint Waypoint (Variable): motionParameters(jointSpeed=1.047198 jointAcceleration=1.396263 cartesianSpeed=0.15 cartesianAcceleration=0.2); variable=PosFinal
                MoveDirectionNode (selectedDirection=ZMinus toolParams=0.02, 0.02)
                  Until DISTANCE (allowActions=false deceleration=3 distanceNodeType=STOP) Distance=0.075; motionParameters(blendRadius=0)
                MoveDirectionNode (selectedDirection=ZPlus toolParams=0.02, 0.02)
                  Until DISTANCE (allowActions=false deceleration=3 distanceNodeType=STOP) Distance=0.075; motionParameters(blendRadius=0)
            Folder Buje26
              Xfin := ((0.73025*Xp)-(Xd)-(0.3937*(1/m2)))*(-1)
              Yfin := ((0.3937*Yp)-(Yd)+(0.73025*m1))*(-1)
              rotaciones := get_actual_tcp_pose()
              var_3 := rotaciones[3]
              var_4 := rotaciones[4]
              var_5 := rotaciones[5]
              PosFinal := p[Xfin+0.00208915,Yfin+0.00208915,-0.44,var_3,var_4,var_5]
              MoveL speed 250 mm/s, acceleration 1200 mm/s^2 (useActiveTCP=true) feature=Base
                MoveJ speed 60 deg/s, acceleration 80 deg/s^2 (useActiveTCP=true) feature=Base
                  Waypoint Waypoint (Variable): motionParameters(jointSpeed=1.047198 jointAcceleration=1.396263 cartesianSpeed=0.15 cartesianAcceleration=0.2); variable=PosFinal
                MoveDirectionNode (selectedDirection=ZMinus toolParams=0.02, 0.02)
                  Until DISTANCE (allowActions=false deceleration=3 distanceNodeType=STOP) Distance=0.075; motionParameters(blendRadius=0)
                MoveDirectionNode (selectedDirection=ZPlus toolParams=0.02, 0.02)
                  Until DISTANCE (allowActions=false deceleration=3 distanceNodeType=STOP) Distance=0.075; motionParameters(blendRadius=0)
            Folder Buje27
              Xfin := ((0.75565*Xp)-(Xd)-(0.3937*(1/m2)))*(-1)
              Yfin := ((0.3937*Yp)-(Yd)+(0.75565*m1))*(-1)
              rotaciones := get_actual_tcp_pose()
              var_3 := rotaciones[3]
              var_4 := rotaciones[4]
              var_5 := rotaciones[5]
              PosFinal := p[Xfin+0.00208915,Yfin+0.00208915,-0.44,var_3,var_4,var_5]
              MoveL speed 250 mm/s, acceleration 1200 mm/s^2 (useActiveTCP=true) feature=Base
                MoveJ speed 60 deg/s, acceleration 80 deg/s^2 (useActiveTCP=true) feature=Base
                  Waypoint Waypoint (Variable): motionParameters(jointSpeed=1.047198 jointAcceleration=1.396263 cartesianSpeed=0.15 cartesianAcceleration=0.2); variable=PosFinal
                MoveDirectionNode (selectedDirection=ZMinus toolParams=0.02, 0.02)
                  Until DISTANCE (allowActions=false deceleration=3 distanceNodeType=STOP) Distance=0.075; motionParameters(blendRadius=0)
                MoveDirectionNode (selectedDirection=ZPlus toolParams=0.02, 0.02)
                  Until DISTANCE (allowActions=false deceleration=3 distanceNodeType=STOP) Distance=0.075; motionParameters(blendRadius=0)
      P5 := p[-0.41462,-0.36474,-0.00863,0,0,0]
      P6 := p[-1.17399,-0.36726,-0.00032,0,0,0]
      P7 := p[-0.38926,-0.09906,-0.00906,0,0,0]
      PQ := pose_sub(P6, P5)
      PR := pose_sub(P7, P5)
      n := p[(PQ[1]*PR[2])-(PQ[2]*PR[1]),(-1)*((PQ[0]*PR[2])-(PQ[2]*PR[0])),(PQ[0]*PR[1])-(PQ[1]*PR[0]),0,0,0]
      var_8 := get_actual_tcp_pose()
      Script: textmsg(Plane_5)
      Popup Message (haltProgram=false inputType=Variable) variable=var_8
    MoveL speed 250 mm/s, acceleration 1200 mm/s^2 (useActiveTCP=true) feature=Plane_5
      MoveDirectionNode (selectedDirection=ZPlus)
        Until DISTANCE (allowActions=false deceleration=3 distanceNodeType=STOP) Distance=0.1; motionParameters(blendRadius=0)
      MoveJ speed 60 deg/s, acceleration 80 deg/s^2 (useActiveTCP=true) feature=Base
        Waypoint casa: TCP in base x=-727.761 y=-161.288 z=455.169 mm, rx=2.012 ry=-2.4053 rz=-0.0107 rad; joints [-1.081, -90.004, 90.001, 0, 90, 0] deg; TCP offset x=0.411 y=-218.298 z=37.994 mm, rx=1.558 ry=-0.1255 rz=0.1212 rad
      MoveL speed 250 mm/s, acceleration 1200 mm/s^2 (useActiveTCP=true) feature=Base
        MoveJ speed 60 deg/s, acceleration 80 deg/s^2 (useActiveTCP=true) feature=Base
          Waypoint Casa2: TCP in base x=-771.144 y=-432.919 z=130.536 mm, rx=2.0101 ry=-2.4029 rz=-0.0102 rad; joints [21.813, -67.428, 96.538, -29.271, 112.826, 0.127] deg; TCP offset x=0.411 y=-218.298 z=37.994 mm, rx=1.558 ry=-0.1255 rz=0.1212 rad
        Folder P1
          Loop While (checkContinuously=false) expression=muestrasTomadas<muestras
            MoveJ speed 60 deg/s, acceleration 80 deg/s^2 (useActiveTCP=true) feature=Base
              Waypoint Sacar_P1: motionParameters(jointSpeed=1.047198 jointAcceleration=1.396263 cartesianSpeed=0.1 cartesianAcceleration=0.15); TCP in base x=-414.573 y=-364.711 z=-6.995 mm, rx=2.0101 ry=-2.4029 rz=-0.0102 rad; joints [31.762, -83.203, 136.491, -53.453, 122.743, 0.135] deg
            Wait Sleep waitTime=0.5
            MoveDirectionNode (selectedDirection=YPlus toolParams=0.0013, 2.0E-4)
              Until TOOL_CONTACT_DETECTION (allowActions=false retraction=0 decelerationAcceleration=9 decelerationAngularAcceleration=34.906585)
            Wait Sleep waitTime=2
            P1 := pose_add(get_actual_tcp_pose(), P1)
            muestrasTomadas := muestrasTomadas+1
          muestrasTomadas := 0
          var_1 := (P1[0])/muestras
          var_2 := (P1[1])/muestras
          rotaciones := get_actual_tcp_pose()
          var_3 := rotaciones[3]
          var_4 := rotaciones[4]
          var_5 := rotaciones[5]
          P1 := p[var_1,var_2,-0.37,var_3,var_4,var_5]
        MoveJ speed 60 deg/s, acceleration 80 deg/s^2 (useActiveTCP=true) feature=Base
          Waypoint Casa2: TCP in base x=-771.144 y=-432.919 z=130.536 mm, rx=2.0101 ry=-2.4029 rz=-0.0102 rad; joints [21.813, -67.428, 96.538, -29.271, 112.826, 0.127] deg
        Folder P2
          Loop While (checkContinuously=false) expression=muestrasTomadas<muestras
            MoveJ speed 60 deg/s, acceleration 80 deg/s^2 (useActiveTCP=true) feature=Base
